PROGRAM UserMode
VAR

(*GapMode*)
	UserGapPositionNew:LREAL:=20;//target
	UserGapVelocityNew:LREAL:=1;//target
	UserGapPositionDisplay:LREAL;//current
	UserGapVelocityDisplay:LREAL;//current
(*ID taper mode*)
	UserTaperPositionNew:LREAL:=0;//target
	UserTaperVelocityNew:LREAL:=0.02;//target
	UserTaperPositionDisplay:LREAL;//current
	UserTaperPositionDisplayBLSide:LREAL;//current BeamLine
	UserTaperPositionActual:LREAL;//current
	UserTaperVelocityDisplay:LREAL;//target
	UserGapPositionDisplay_FromLeftTop:LREAL;
	UserGapPositionDisplay_FromLeftBottom:LREAL;
		//
	UserRightGapPositionNew:LREAL;
	UserRightGapVelocityNew:LREAL;
	UserRightGapPositionDisplay:LREAL;
	UserRightGapVelocityDisplay:LREAL;
	UserRightGapPositionDisplay_FromRightTop:LREAL;
	UserRightGapPositionDisplay_FromRightBottom:LREAL;
(*BL taper mode*)
	BLUserTaperPositionNew:LREAL:=0;//target
	BLUserTaperVelocityNew:LREAL:=0.02;//target
	BLUserTaperPositionDisplay:LREAL;//current
	//BLUserTaperPositionDisplayBLSide:LREAL;//current BeamLine
	BLUserTaperPositionActual:LREAL;//current
	BLUserTaperVelocityDisplay:LREAL;//target
	BLUserGapPositionDisplay_FromLeftTop:LREAL;
	BLUserGapPositionDisplay_FromLeftBottom:LREAL;
	//
	BLUserLeftGapPositionNew:LREAL;
	BLUserLeftGapVelocityNew:LREAL;
	BLUserLeftGapPositionDisplay:LREAL;
	BLUserLeftGapVelocityDisplay:LREAL;
	BLUserLeftGapPositionDisplay_FromLeftTop:LREAL;
	BLUserLeftGapPositionDisplay_FromLeftBottom:LREAL;
	BLUserRightGapPositionNew:LREAL;
	BLUserRightGapVelocityNew:LREAL;
	BLUserRightGapPositionDisplay:LREAL;
	BLUserRightGapVelocityDisplay:LREAL;
	BLUserRightGapPositionDisplay_FromRightTop:LREAL;
	BLUserRightGapPositionDisplay_FromRightBottom:LREAL;
(*PhaseUpper Move*)
	UserPhaseUpperPositionNew:LREAL:=0;//target
	UserPhaseUpperVelocityNew:LREAL:=0.5;//target
(*PhaseUpper Move*)
	UserPhaseLowerPositionNew:LREAL:=0;//target
	UserPhaseLowerVelocityNew:LREAL:=0.5;//target
	UserPhaseLowerPositionDisplay:LREAL;//current
	UserPhaseLowerVelocityDisplay:LREAL;//current
	//
	(*Gap move&Stop*)
	btn_UserGapMove:BOOL;
	btn_UserGapStop:BOOL;
	(*PhaseUpper Move&Stop*)
	btn_UserPhaseUpperMove:BOOL;
	btn_UserPhaseUpperStop:BOOL;
	(*PhaseLower Move&Stop*)
	btn_UserPhaseLowerMove:BOOL;
	btn_UserPhaseLowerStop:BOOL;
	(*Var*)
	fb_ton1:TON;
	fb_ton2:TON;
	fb_ton3:TON;
	fb_ton4:TON;
	fb_ton5:TON;
	fb_ton6:TON;
	(*Status*)
	State:DINT;
	Busy:BOOL;
	InitPowerDone:BOOL;
	InitCompensationDatasDone:BOOL;
	(*FB*)
	m_state: DINT;
	n_state: DINT;
	s_state: DINT;
	m_state_PhaseUpper: DINT;
	n_state_PhaseUpper: DINT;
	s_state_PhaseUpper: DINT;
	m_state_PhaseLower: DINT;
	n_state_PhaseLower: DINT;
	s_state_PhaseLower: DINT;
	(*¼ì²âµ½ÏÞÎ»£¬»Ö¸´Move×´Ì¬*)
	FTrig_ReachLS: F_TRIG;
	FTrig_ReachLS_PhaseUpper: F_TRIG;
	FTrig_ReachLS_PhaseLower: F_TRIG;
	FTrig_btn_GapMove: F_TRIG;
	GapOutRange: BOOL;
	(*PowerOff*)
	d_state: DINT;
	i: INT;
	j: INT;
	k: INT;
	moni_State:DINT;
	TargetPosLessThanCurrentPos:BOOL;
	TargetLTPosLessThanCurrentLTPos:BOOL;
	TargetRTPosLessThanCurrentRTPos:BOOL;
	TargetLBPosLessThanCurrentLBPos:BOOL;
	TargetRBPosLessThanCurrentRBPos:BOOL;
	PositiveMoving:BOOL;
	HysteresisMoving:BOOL;
	NoneHysteresisMoving:BOOL;
	(**)
	TargetPosLessThanCurrentPos_PhaseUpper:BOOL;
	PositiveMoving_PhaseUpper:BOOL;
	HysteresisMoving_PhaseUpper:BOOL;
	NoneHysteresisMoving_PhaseUpper:BOOL;
	TargetPosLessThanCurrentPos_PhaseLower:BOOL;
	PositiveMoving_PhaseLower:BOOL;
	HysteresisMoving_PhaseLower:BOOL;
	NoneHysteresisMoving_PhaseLower:BOOL;
	(*Spectroscopy scanning Mode*)
	IsSSMotionMode:BOOL;
	RegularMotionMode:BOOL;
	SSMotionMode:BOOL;
	SS_StepSize:LREAL:=0.001;
	SS_StepNumber:INT:=10;
	SS_StepVelocity:LREAL:=1;
	SS_Move:BOOL;
	SS_Stop:BOOL;
	SS_MoveState:DINT;
	SS_StopState:DINT;
	SS_currentStep:DINT:=0;
	SS_StepSystemTime_Begin:ARRAY[0..100] OF ULINT;
	SS_StepSystemTime_End:ARRAY[0..100] OF ULINT;
	SS_StepCountTime:ARRAY[0..100] OF ULINT;
	SS_TimeCountBegin:BOOL;
	m: INT;
	SS_TON: TON;
	StepEachTime:TIME;
	StepEachTime_ms:INT:=1000;//ms
	SS_OTSTRUCT :OTSTRUCT ;
	SS_StartPositionDisplay:LREAL;
	RTRG_SS_StartPositionDisplay:R_TRIG;
	SS_InitStartPositionDone:BOOL;
	
	//
	min_SS_StepSize	: LREAL:=0;
	max_SS_StepSize	: LREAL:=200;
	inRange_SS_StepSize	: BOOL;
	//
	min_SS_StepNumber	: INT:=1;
	max_SS_StepNumber	: INT:=1000;
	inRange_SS_StepNumber	: BOOL;
	//
	min_SS_StepVelocity:LREAL:=0;
	max_SS_StepVelocity:LREAL:=1;
	inRange_SS_StepVelocity:BOOL;
	//
	min_StepEachTime_ms:INT:=100;
	max_StepEachTime_ms:INT:=10000;
	inRange_StepEachTime_ms:BOOL;
	l: INT;
	Threshold_UserTopPos_PLC: LREAL;
	Threshold_UserTopVelo_PLC: LREAL;
	Threshold_UserBottomPos_PLC: LREAL;
	Threshold_UserBottomVelo_PLC: LREAL;
	Threshold_UserLeftPos_PLC: LREAL;
	Threshold_UserLeftVelo_PLC: LREAL;
	Threshold_UserRightPos_PLC: LREAL;
	Threshold_UserRightVelo_PLC: LREAL;
	testa: BOOL;
	testb: BOOL;
	Threshold_GapChangeFlag: LREAL;
	Threshold_TaperChangeFlag: LREAL;
	TaperAndGapSafetyfactor: LREAL:=1;
	//GapPhase Chain protection
	GapPhase_ChainProtection_On:BOOL;
	GapPhase_ChainProtection_MaxGapValue: LREAL;
	//
	//Global Chain protection-MPS
	Global_ChainProtection_MPS_StorageRingReady:BOOL;
	Global_ChainProtection_MPS_On: BOOL;
	Global_ChainProtection_MPS_MaxGapValue: LREAL;
	Global_ChainProtection_MPS_MoveVelocity: LREAL;
	Global_ChainProtection_MPS_Done: BOOL;
	//Global_ChainProtection_Error: BOOL;
	//Global_ChainProtection_ErrorID: INT;
	//Global_ChainProtection_ErrorDescription: STRING;
	Global_ChainProtection_MPS_ManualOperation:BOOL:=TRUE;
	Global_ChainProtection_MPS_FTRIG:F_TRIG;
	Global_ChainProtection_MPS_FTRIG_Manul:F_TRIG;
	Global_ChainProtection_MPS_TON:TON;
	Global_ChainProtection_MPS_Triggered:BOOL;
	Global_ChainProtection_MPS_In:BOOL;
	Global_ChainProtection_MPS_In1 AT%I* :BOOL;//下降沿表示触发,EL1008
	Global_ChainProtection_MPS_In2 AT%I* :BOOL;
	Global_ChainProtection_MPS_State:DINT;
	Global_ChainProtection_MPS_Out1 AT%Q* :BOOL;//上升沿标识到达最大间隙，连锁保护成功,EL2624
	Global_ChainProtection_MPS_Out2 AT%Q* :BOOL;
	Global_ChainProtection_MPS_TON_Stop2Move:TON;
	Global_ChainProtection_MPS_TON_Stop2Move_InTaperMode:TON;
	Global_ChainProtection_MPS_TON_Power2Move:TON;
	//Global Chain protection-EPS
	Global_ChainProtection_EPS_BeamLineReady:BOOL;
	Global_ChainProtection_EPS_On: BOOL;
	Global_ChainProtection_EPS_MaxGapValue: LREAL;
	Global_ChainProtection_EPS_MoveVelocity: LREAL;
	Global_ChainProtection_EPS_Done: BOOL;
	//Global_ChainProtection_Error: BOOL;
	//Global_ChainProtection_ErrorID: INT;
	//Global_ChainProtection_ErrorDescription: STRING;
	Global_ChainProtection_EPS_ManualOperation:BOOL:=TRUE;
	Global_ChainProtection_EPS_FTRIG:F_TRIG;
	Global_ChainProtection_EPS_FTRIG_Manul:F_TRIG;
	Global_ChainProtection_EPS_TON:TON;
	Global_ChainProtection_EPS_Triggered:BOOL;
	Global_ChainProtection_EPS_In:BOOL;
	Global_ChainProtection_EPS_In1 AT%I* :BOOL;//下降沿表示触发,EL1124
	Global_ChainProtection_EPS_In2 AT%I* :BOOL;
	Global_ChainProtection_EPS_State:DINT;
	Global_ChainProtection_EPS_Out1 AT%Q* :BOOL;//上升沿标识到达最大间隙，连锁保护成功,EL2124
	Global_ChainProtection_EPS_Out2 AT%Q* :BOOL;
	Global_ChainProtection_EPS_TON_Stop2Move:TON;
	Global_ChainProtection_EPS_TON_Stop2Move_InTaperMode:TON;
	Global_ChainProtection_EPS_TON_Power2Move:TON;
	
	Threshold_motorsTargetPosCalculate: LREAL;
	LeftTopLinPositionNewTemp: LREAL;
	RightTopLinPositionNewTemp: LREAL;
	LeftBottomLinPositionNewTemp: LREAL;
	RightBottomLinPositionNewTemp: LREAL;
	UserPhaseUpperPositionNewTemp: LREAL;
	UserPhaseLowerPositionNewTemp: LREAL;
	
	//OneKeyToMaxGap
	btn_OneKeyToMaxGap:BOOL;
	OneKeyToMaxGap_RTRIG:R_TRIG;
	OneKeyToMaxGap_TON:TON;
	OneKeyToMaxGap_Triggered:BOOL;
	OneKeyToMaxGap_State:DINT;
	OneKeyToMaxGap_TON_Stop2Move:TON;
	OneKeyToMaxGap_TON_Stop2Move_InTaperMode:TON;
	OneKeyToMaxGap_TON_Power2Move:TON;
	OneKeyToMaxGap_Done:BOOL;
	
		//BLTaper
	CurrentTaperInit: LREAL;
	L_HalfGirder:LREAL:=2500;
	L_Center2Motor:LREAL:=1375;
	//
	trig_TaperOrNot: R_TRIG;
	trig_BLTaperOrNot: R_TRIG;
	
	//
	//零位特殊走法
	//
	(*Upper*)
    // 零位特殊走法总开关。TRUE 启用；FALSE 关闭，关闭后直接按原 m/n 正常逻辑运行。
    EnableZeroPre_PhaseUpper : BOOL := TRUE;

    // 判断“当前位置在零附近”的范围。例如当前位置绝对值 <= 0.01mm 认为在零附近。
    ZeroNearThreshold_PhaseUpper : LREAL := 0.3;

    // 原来的 +/-1mm 边界，做成变量，后续可以改成 +/-0.5mm、+/-2mm 等。
    ZeroBoundary_PhaseUpper : LREAL := 1.5;

    // 零位附近特殊慢速，原来的 0.1mm/s，做成变量。
    ZeroSlowVelocity_PhaseUpper : LREAL := 0.1;

    // TRUE 表示当前正在执行零位预走状态机，此时屏蔽原 m/n 正常逻辑。
    ZeroPreMoving_PhaseUpper : BOOL := FALSE;

    // TRUE 表示本次 Move 的零位预走已经完成，下一步允许进入原 m/n 正常逻辑；正常完成或 Stop 时必须清 FALSE。
    ZeroPreDone_PhaseUpper : BOOL := FALSE;

    // TRUE 表示目标就在 +/-ZeroBoundary_PhaseUpper 内，此时只需要慢速直接走到目标，不再进入原 m/n 正常逻辑。
    ZeroDirectMove_PhaseUpper : BOOL := FALSE;

    // 零位预走专用状态。
    z_state_PhaseUpper : INT := 0;

    // 零位预走第一段目标：目标超过边界时为 +ZeroBoundary/-ZeroBoundary；目标在边界内时为最终目标。
    ZeroPreTarget_PhaseUpper : LREAL := 0.0;

    // 锁存本次 Move 的最终目标，避免零位慢速段期间用户改输入导致最终目标漂移。
    ZeroFinalTarget_PhaseUpper : LREAL := 0.0;

    // 锁存本次 Move 的用户速度，零位预走之后原 m/n 逻辑使用这个速度。
    ZeroFinalVelocity_PhaseUpper : LREAL := 0.0;

    // 原 m/n 正常逻辑当前使用的目标；零位预走后用 ZeroFinalTarget_PhaseUpper，否则用 UserPhaseUpperPositionNew。
    ActiveTarget_PhaseUpper : LREAL := 0.0;

    // 原 m/n 正常逻辑当前使用的速度；零位预走后用 ZeroFinalVelocity_PhaseUpper，否则用 UserPhaseUpperVelocityNew。
    ActiveVelocity_PhaseUpper : LREAL := 0.0;
	
	(*Lower*)
	
    // 零位特殊走法总开关。TRUE 启用；FALSE 关闭，关闭后直接按原 m/n 正常逻辑运行。
    EnableZeroPre_PhaseLower : BOOL := TRUE;

    // 判断“当前位置在零附近”的范围。例如当前位置绝对值 <= 0.01mm 认为在零附近。
    ZeroNearThreshold_PhaseLower : LREAL := 0.3;

    // 原来的 +/-1mm 边界，做成变量，后续可以改成 +/-0.5mm、+/-2mm 等。
    ZeroBoundary_PhaseLower : LREAL := 1.5;

    // 零位附近特殊慢速，原来的 0.1mm/s，做成变量。
    ZeroSlowVelocity_PhaseLower : LREAL := 0.1;

    // TRUE 表示当前正在执行零位预走状态机，此时屏蔽原 m/n 正常逻辑。
    ZeroPreMoving_PhaseLower : BOOL := FALSE;

    // TRUE 表示本次 Move 的零位预走已经完成，下一步允许进入原 m/n 正常逻辑；正常完成或 Stop 时必须清 FALSE。
    ZeroPreDone_PhaseLower : BOOL := FALSE;

    // TRUE 表示目标就在 +/-ZeroBoundary_PhaseLower 内，此时只需要慢速直接走到目标，不再进入原 m/n 正常逻辑。
    ZeroDirectMove_PhaseLower : BOOL := FALSE;

    // 零位预走专用状态。
    z_state_PhaseLower : INT := 0;

    // 零位预走第一段目标：目标超过边界时为 +ZeroBoundary/-ZeroBoundary；目标在边界内时为最终目标。
    ZeroPreTarget_PhaseLower : LREAL := 0.0;

    // 锁存本次 Move 的最终目标，避免零位慢速段期间用户改输入导致最终目标漂移。
    ZeroFinalTarget_PhaseLower : LREAL := 0.0;

    // 锁存本次 Move 的用户速度，零位预走之后原 m/n 逻辑使用这个速度。
    ZeroFinalVelocity_PhaseLower : LREAL := 0.0;

    // 原 m/n 正常逻辑当前使用的目标；零位预走后用 ZeroFinalTarget_PhaseLower，否则用 UserPhaseLowerPositionNew。
    ActiveTarget_PhaseLower : LREAL := 0.0;

    // 原 m/n 正常逻辑当前使用的速度；零位预走后用 ZeroFinalVelocity_PhaseLower，否则用 UserPhaseLowerVelocityNew。
    ActiveVelocity_PhaseLower : LREAL := 0.0;
 
	
END_VAR

IF NOT PositionBiasDone THEN
	RETURN;
END_IF
IF NOT loadParametersDone THEN
	RETURN;
END_IF
(*btn_Power On/Off*)
IF btn_Power AND st_Power=0 THEN
	btn_PowerOn:=TRUE;
	btn_Power:=FALSE;
END_IF
IF btn_Power AND st_Power=1 THEN
	btn_PowerOff:=TRUE;
	btn_Power:=FALSE;
END_IF
IF btn_PowerOn THEN
	A_PowerOn();
END_IF
IF btn_PowerOff THEN
	A_PowerOff();
END_IF

(*检查couple状态，不允许couple*)
A_CheckCoupleStatus();

(*监控四轴位置速度等*)
A_MonitoringAllAxis();

(*补偿数据处理*)
A_InitCompensationData();

(*目标位置和速度保护*)
A_CheckMotorsPos();


(*常规磁间隙开合*)
//IF RegularMotionMode AND NOT SSMotionMode THEN
A_RegularMotion();
//END_IF
(*PhaseUpper运动*)
A_PhaseUpperMotion();
(*PhaseLower运动*)
A_PhaseLowerMotion();
(*Spectroscopy scanning Mode*)
IF IsSSMotionMode THEN
	SSMotionMode:=TRUE;
	RegularMotionMode:=FALSE;
ELSE
	SSMotionMode:=FALSE;
	RegularMotionMode:=TRUE;
END_IF
IF	SSMotionMode AND NOT RegularMotionMode THEN
	A_SpectroscopyScanningMotion();
END_IF
(*GlobalChainProtection*)
A_GlobalChainProtection_EPS();
A_GlobalChainProtection_MPS();
(*A_OneKeyToMaxGap*)
A_OneKeyToMaxGap();

ACTION A_CheckCoupleStatus:
IF NOT btn_PowerOff THEN
	IF st_Power=1 AND st_Couple<>0THEN
		Error:=TRUE;
		ErrorID:=501;
		LeftTopLinMoveIndicator:=0;
		RightTopLinMoveIndicator:=0;
		LeftBottomLinMoveIndicator:=0;
		RightBottomLinMoveIndicator:=0;
		FB_PlcEmergencyStop();
		LED_Error:=TRUE;
		ErrorDescription:='couple stutas error';
	END_IF
END_IF
END_ACTION

ACTION A_CheckMotorsPos:
//
//目标位置速度超出阈值判断
//
//gap posiion
IF UserGapPositionNew<min_UserGapPositionNew OR UserGapPositionNew>max_UserGapPositionNew THEN
	inRange_UserGapPositionNew:=FALSE;
END_IF
IF UserGapPositionNew>=min_UserGapPositionNew AND UserGapPositionNew<=max_UserGapPositionNew THEN
	inRange_UserGapPositionNew:=TRUE;
END_IF
//gap velocity
IF UserGapVelocityNew<min_UserGapVelocityNew OR UserGapVelocityNew>max_UserGapVelocityNew THEN
	inRange_UserGapVelocityNew:=FALSE;
END_IF
IF UserGapVelocityNew>=min_UserGapVelocityNew AND UserGapVelocityNew<=max_UserGapVelocityNew THEN
	inRange_UserGapVelocityNew:=TRUE;
END_IF
//taper position
IF UserTaperPositionNew<min_UserTaperPositionNew OR UserTaperPositionNew>max_UserTaperPositionNew THEN
	inRange_UserTaperPositionNew:=FALSE;
END_IF
IF UserTaperPositionNew>=min_UserTaperPositionNew AND UserTaperPositionNew<=max_UserTaperPositionNew THEN
	inRange_UserTaperPositionNew:=TRUE;
END_IF
//taper velocity
IF UserTaperVelocityNew<min_UserTaperVelocityNew OR UserTaperVelocityNew>max_UserTaperVelocityNew THEN
	inRange_UserTaperVelocityNew:=FALSE;
END_IF
IF UserTaperVelocityNew>=min_UserTaperVelocityNew AND UserTaperVelocityNew<=max_UserTaperVelocityNew THEN
	inRange_UserTaperVelocityNew:=TRUE;
END_IF
//
//PhaseUpper posiion
IF UserPhaseUpperPositionNew<min_UserPhaseUpperPositionNew OR UserPhaseUpperPositionNew>max_UserPhaseUpperPositionNew THEN
	inRange_UserPhaseUpperPositionNew:=FALSE;
END_IF
IF UserPhaseUpperPositionNew>=min_UserPhaseUpperPositionNew AND UserPhaseUpperPositionNew<=max_UserPhaseUpperPositionNew THEN
	inRange_UserPhaseUpperPositionNew:=TRUE;
END_IF
//gap velocity
IF UserPhaseUpperVelocityNew<min_UserPhaseUpperVelocityNew OR UserPhaseUpperVelocityNew>max_UserPhaseUpperVelocityNew THEN
	inRange_UserPhaseUpperVelocityNew:=FALSE;
END_IF
IF UserPhaseUpperVelocityNew>=min_UserPhaseUpperVelocityNew AND UserPhaseUpperVelocityNew<=max_UserPhaseUpperVelocityNew THEN
	inRange_UserPhaseUpperVelocityNew:=TRUE;
END_IF
//PhaseLower posiion
IF UserPhaseLowerPositionNew<min_UserPhaseLowerPositionNew OR UserPhaseLowerPositionNew>max_UserPhaseLowerPositionNew THEN
	inRange_UserPhaseLowerPositionNew:=FALSE;
END_IF
IF UserPhaseLowerPositionNew>=min_UserPhaseLowerPositionNew AND UserPhaseLowerPositionNew<=max_UserPhaseLowerPositionNew THEN
	inRange_UserPhaseLowerPositionNew:=TRUE;
END_IF
//gap velocity
IF UserPhaseLowerVelocityNew<min_UserPhaseLowerVelocityNew OR UserPhaseLowerVelocityNew>max_UserPhaseLowerVelocityNew THEN
	inRange_UserPhaseLowerVelocityNew:=FALSE;
END_IF
IF UserPhaseLowerVelocityNew>=min_UserPhaseLowerVelocityNew AND UserPhaseLowerVelocityNew<=max_UserPhaseLowerVelocityNew THEN
	inRange_UserPhaseLowerVelocityNew:=TRUE;
END_IF
//SS Mode
IF SS_StepSize<min_SS_StepSize OR SS_StepSize>max_SS_StepSize THEN
	inRange_SS_StepSize:=FALSE;
END_IF
IF SS_StepSize>=min_SS_StepSize AND SS_StepSize<=max_SS_StepSize THEN
	inRange_SS_StepSize:=TRUE;
END_IF
IF SS_StepNumber<min_SS_StepNumber OR SS_StepNumber>max_SS_StepNumber THEN
	inRange_SS_StepNumber:=FALSE;
END_IF
IF SS_StepNumber>=min_SS_StepNumber AND SS_StepNumber<=max_SS_StepNumber THEN
	inRange_SS_StepNumber:=TRUE;
END_IF
IF SS_StepVelocity<min_SS_StepVelocity OR SS_StepVelocity>max_SS_StepVelocity THEN
	inRange_SS_StepVelocity:=FALSE;
END_IF
IF SS_StepVelocity>=min_SS_StepVelocity AND SS_StepVelocity<=max_SS_StepVelocity THEN
	inRange_SS_StepVelocity:=TRUE;
END_IF
IF StepEachTime_ms<min_StepEachTime_ms OR StepEachTime_ms>max_StepEachTime_ms THEN
	inRange_StepEachTime_ms:=FALSE;
END_IF
IF StepEachTime_ms>=min_StepEachTime_ms AND StepEachTime_ms<=max_StepEachTime_ms THEN
	inRange_StepEachTime_ms:=TRUE;
END_IF


//
//输入速度和位置保护
//
IF btn_UserGapMove  AND NOT SSMotionMode AND RegularMotionMode THEN
	IF NOT inRange_UserGapPositionNew THEN
		btn_UserGapStop:=TRUE;
		btn_UserGapMove:=FALSE;
		Error:=TRUE;
		ErrorId:=801;
		ErrorDescription:='target Gap position out of range,please check';
		RETURN;
	ELSE
		//btn_UserGapStop:=FALSE;
		Error:=FALSE;
		ErrorId:=0;
		ErrorDescription:='';	
	END_IF
	IF NOT inRange_UserGapVelocityNew THEN
		btn_UserGapStop:=TRUE;
		btn_UserGapMove:=FALSE;
		Error:=TRUE;
		ErrorId:=802;
		ErrorDescription:='target Gap velocity out of range,please check';
		RETURN;
	ELSE
		//btn_UserGapStop:=FALSE;
		Error:=FALSE;
		ErrorId:=0;
		ErrorDescription:='';
	END_IF
END_IF

//
//运动过程中，监控目标位置速度
//
IF moveStatusAnyAxis THEN
	IF NOT inRange_UserGapPositionNew THEN
		btn_UserGapStop:=TRUE;
		Error:=TRUE;
		ErrorId:=805;
		ErrorDescription:='target Gap position out of range in moving process!';
		FB_PlcEmergencyStop();
	END_IF
	IF NOT inRange_UserGapVelocityNew THEN
		btn_UserGapStop:=TRUE;
		Error:=TRUE;
		ErrorId:=806;
		ErrorDescription:='target Gap velocity out of range in moving process!';
		FB_PlcEmergencyStop();
	END_IF
END_IF
//
//运动过程中，监控每一个轴的目标位置，目标位置若超出阈值，Emergency
//
IF moveStatusAnyAxis THEN
	IF NOT TaperOrNot THEN
		IF LeftTopLinPositionNew<min_UserLEProtectionGapPosition/2 OR LeftTopLinPositionNew>max_UserLEProtectionGapPosition/2 THEN
			btn_UserGapStop:=TRUE;
			Error:=TRUE;
			ErrorId:=809;
			ErrorDescription:='target LeftTop position out of range in moving process!';
			FB_PlcEmergencyStop();
		END_IF
		IF RightTopLinPositionNew<min_UserLEProtectionGapPosition/2 OR RightTopLinPositionNew>max_UserLEProtectionGapPosition/2 THEN
			btn_UserGapStop:=TRUE;
			Error:=TRUE;
			ErrorId:=810;
			ErrorDescription:='target RightTop velocity out of range in moving process!';
			FB_PlcEmergencyStop();
		END_IF
		IF LeftBottomLinPositionNew<min_UserLEProtectionGapPosition/2 OR LeftBottomLinPositionNew>max_UserLEProtectionGapPosition/2 THEN
			btn_UserGapStop:=TRUE;
			Error:=TRUE;
			ErrorId:=812;
			ErrorDescription:='target LeftBottom Position out of range in moving process!';
			FB_PlcEmergencyStop();
		END_IF
		IF RightBottomLinPositionNew<min_UserLEProtectionGapPosition/2 OR RightBottomLinPositionNew>max_UserLEProtectionGapPosition/2 THEN
			btn_UserGapStop:=TRUE;
			Error:=TRUE;
			ErrorId:=813;
			ErrorDescription:='target RightBottom Position out of range in moving process!';
			FB_PlcEmergencyStop();
		END_IF
	ELSE//Taper状态的保护
		;//Taper状态下，不用监控四轴位置，只需要监控目标Taper位置。在上面已经保护
	END_IF
END_IF
END_ACTION

ACTION A_GlobalChainProtection_EPS:
//硬线输入定义
Global_ChainProtection_EPS_In:=Global_ChainProtection_EPS_In1 AND Global_ChainProtection_EPS_In2;
//硬线输出定义
Global_ChainProtection_EPS_Out1:=Global_ChainProtection_EPS_Done;
Global_ChainProtection_EPS_Out2:=Global_ChainProtection_EPS_Done;
//总开关
IF NOT Global_ChainProtection_EPS_On THEN
	RETURN;
END_IF
//判断插入件状态，是否就位
//IF NOT IDControlReady THEN
//	Global_ChainProtection_EPS_Done:=FALSE;
//	Error:= TRUE;
//	ErrorID:= 1501;
//	ErrorDescription:='ID NOT READY!';
//	RETURN;
//END_IF
//判断储存环是否给出就位信号，暂时由参数表给出TRUE，最终将由IOC接受PV
IF 	NOT Global_ChainProtection_EPS_BeamLineReady THEN
	Global_ChainProtection_EPS_Done:=FALSE;
	Error:= TRUE;
	ErrorID:= 1503;
	ErrorDescription:='Global_ChainProtection_EPS_BeamLineReady NOT Ready';
	RETURN;
END_IF
//
//全局连锁保护程序开始
//
//0.检测到下降沿，触发
//1.判断电机是否在开启状态,没有就打开电源
//2.判断是否在Moving状态,若有就Stop
//3.将磁间隙打开到至最大阈值
//4.到位后给出反馈，且安全PLC触发
Global_ChainProtection_EPS_FTRIG(CLK:=Global_ChainProtection_EPS_In);
IF Global_ChainProtection_EPS_FTRIG.Q THEN
	Global_ChainProtection_EPS_Triggered:=TRUE;
END_IF
Global_ChainProtection_EPS_FTRIG_Manul(CLK:=Global_ChainProtection_EPS_ManualOperation);
IF Global_ChainProtection_EPS_FTRIG_Manul.Q THEN
	Global_ChainProtection_EPS_Triggered:=TRUE;
END_IF
IF Global_ChainProtection_EPS_Triggered THEN
	CASE Global_ChainProtection_EPS_State OF
		0://1.判断电机是否在开启状态,没有就打开电源
			IF st_Power=1 THEN
				Global_ChainProtection_EPS_State:=1;
			ELSE
				btn_PowerOn:=TRUE;
				IF btn_PowerOn THEN
					A_PowerOn();
				END_IF
			END_IF
		1://1.判断是否在谱学扫描模式，如果是，则切换回正常运动模式
			IF IsSSMotionMode THEN
				SS_Stop:=TRUE;
				IsSSMotionMode:=FALSE;
			END_IF
			Global_ChainProtection_EPS_State:=2;
		2://判断是否在taper，如果在taper,则判断是否在运动，如果是，则停止运动,0.5sh后，转入下一步
			IF TaperOrNot THEN
				IF moveStatusLeftTop OR moveStatusRightTop OR moveStatusLeftBottom OR moveStatusRightBottom THEN
					btn_UserGapStop:=TRUE;
				ELSE
					Global_ChainProtection_EPS_TON_Stop2Move_InTaperMode(PT:=T#0.5S);
					Global_ChainProtection_EPS_TON_Stop2Move_InTaperMode.IN:=TRUE;
					IF Global_ChainProtection_EPS_TON_Stop2Move_InTaperMode.Q THEN
						TaperOrNot:=FALSE;//关闭taper模式
						Global_ChainProtection_EPS_State:=3;
					END_IF
				END_IF
			ELSE
				Global_ChainProtection_EPS_State:=3;
			END_IF
		3://3.判断是否在Moving状态,若有就Stop.Taper模式已处理完，此处开始走正常GAP开合逻辑
			IF moveStatusLeftTop OR moveStatusRightTop OR moveStatusLeftBottom OR moveStatusRightBottom THEN
				btn_UserGapStop:=TRUE;
			ELSE
				Global_ChainProtection_EPS_TON_Stop2Move(PT:=T#0.5S);
				Global_ChainProtection_EPS_TON_Stop2Move.IN:=TRUE;
				IF Global_ChainProtection_EPS_TON_Stop2Move.Q THEN
					Global_ChainProtection_EPS_State:=4;
				END_IF
			END_IF
		4://当前磁间隙如何和最大磁间隙差别不大，不超过0.1，则直接保护
			IF ABS(UserGapPositionDisplay-Global_ChainProtection_EPS_MaxGapValue)<=0.1 THEN
				Global_ChainProtection_EPS_Done:=TRUE;
				Plc_EmergencyStop:=FALSE;	
				Error:=TRUE;
				ErrorID:=1506;
				ErrorDescription:='EPS Triggered,but ABS(UserGapPositionDisplay-Global_ChainProtection_EPS_MaxGapValue)<=0.1 ';	
			ELSE
				Global_ChainProtection_EPS_State:=5;
			END_IF
		5://5.将磁间隙打开到至最大阈值
			Global_ChainProtection_EPS_TON(PT:=INT_TO_TIME(LREAL_TO_INT(Global_ChainProtection_EPS_MaxGapValue/Global_ChainProtection_EPS_MoveVelocity+30))*1000);
			Global_ChainProtection_EPS_TON.IN:=TRUE;
			Global_ChainProtection_EPS_TON_Power2Move(PT:=T#0.1S);
			Global_ChainProtection_EPS_TON_Power2Move.IN:=TRUE;
			UserGapPositionNew:=Global_ChainProtection_EPS_MaxGapValue;
			UserGapVelocityNew:=Global_ChainProtection_EPS_MoveVelocity;
			btn_UserGapMove:=TRUE;
			IF Global_ChainProtection_EPS_TON_Power2Move.Q THEN
				IF FB_MOVE.BCGapDone THEN
					Global_ChainProtection_EPS_State:=88;
				END_IF
			END_IF
			IF Global_ChainProtection_EPS_TON.Q THEN//如果150s后，还没有运动到指定gap，则报错
				Global_ChainProtection_EPS_State:=-100;
			END_IF
		88://6.到位后给出反馈，且安全PLC触发
			Global_ChainProtection_EPS_Done:=TRUE;
			Plc_EmergencyStop:=FALSE;	
			Error:=TRUE;
			ErrorID:=1504;
			ErrorDescription:='Global_ChainProtection_EPS Triggered ';	
		-100:
			Global_ChainProtection_EPS_Done:=FALSE;
			Error:=TRUE;
			ErrorID:=1505;
			ErrorDescription:='NOT MOVING TO MAXGAP';
	END_CASE
END_IF
END_ACTION

ACTION A_GlobalChainProtection_MPS:
//硬线输入定义
Global_ChainProtection_MPS_In:=Global_ChainProtection_MPS_In1 AND Global_ChainProtection_MPS_In2;
//硬线输出定义
Global_ChainProtection_MPS_Out1:=Global_ChainProtection_MPS_Done;
Global_ChainProtection_MPS_Out2:=Global_ChainProtection_MPS_Done;
//总开关
IF NOT Global_ChainProtection_MPS_On THEN
	RETURN;
END_IF
//判断插入件状态，是否就位
//IF NOT IDControlReady THEN
//	Global_ChainProtection_MPS_Done:=FALSE;
//	Error:= TRUE;
//	ErrorID:= 1401;
//	ErrorDescription:='ID NOT READY!';
//	RETURN;
//END_IF
//判断储存环是否给出就位信号，暂时由参数表给出TRUE，最终将由IOC接受PV
IF 	NOT Global_ChainProtection_MPS_StorageRingReady THEN
	Global_ChainProtection_MPS_Done:=FALSE;
	Error:= TRUE;
	ErrorID:= 1403;
	ErrorDescription:='StorageRingChainProtection NOT Ready';
	RETURN;
END_IF
//
//全局连锁保护程序开始
//
//0.检测到下降沿，触发
//1.判断电机是否在开启状态,没有就打开电源
//2.判断是否在Moving状态,若有就Stop
//3.将磁间隙打开到至最大阈值
//4.到位后给出反馈，且安全PLC触发
Global_ChainProtection_MPS_FTRIG(CLK:=Global_ChainProtection_MPS_In);
IF Global_ChainProtection_MPS_FTRIG.Q THEN
	Global_ChainProtection_MPS_Triggered:=TRUE;
END_IF
Global_ChainProtection_MPS_FTRIG_Manul(CLK:=Global_ChainProtection_MPS_ManualOperation);
IF Global_ChainProtection_MPS_FTRIG_Manul.Q THEN
	Global_ChainProtection_MPS_Triggered:=TRUE;
END_IF
IF Global_ChainProtection_MPS_Triggered THEN
	CASE Global_ChainProtection_MPS_State OF
		0://1.判断电机是否在开启状态,没有就打开电源
			IF st_Power=1 THEN
				Global_ChainProtection_MPS_State:=1;
			ELSE
				btn_PowerOn:=TRUE;
				IF btn_PowerOn THEN
					A_PowerOn();
				END_IF
			END_IF
		1://1.判断是否在谱学扫描模式，如果是，则切换回正常运动模式
			IF IsSSMotionMode THEN
				SS_Stop:=TRUE;
				IsSSMotionMode:=FALSE;
			END_IF
			Global_ChainProtection_MPS_State:=2;
		2://判断是否在taper，如果在taper,则判断是否在运动，如果是，则停止运动,0.5sh后，转入下一步
			IF TaperOrNot THEN
				IF moveStatusLeftTop OR moveStatusRightTop OR moveStatusLeftBottom OR moveStatusRightBottom THEN
					btn_UserGapStop:=TRUE;
				ELSE
					Global_ChainProtection_MPS_TON_Stop2Move_InTaperMode(PT:=T#0.5S);
					Global_ChainProtection_MPS_TON_Stop2Move_InTaperMode.IN:=TRUE;
					IF Global_ChainProtection_MPS_TON_Stop2Move_InTaperMode.Q THEN
						TaperOrNot:=FALSE;//关闭taper模式
						Global_ChainProtection_MPS_State:=3;
					END_IF
				END_IF
			ELSE
				Global_ChainProtection_MPS_State:=3;
			END_IF
		3://3.判断是否在Moving状态,若有就Stop.Taper模式已处理完，此处开始走正常GAP开合逻辑
			IF moveStatusLeftTop OR moveStatusRightTop OR moveStatusLeftBottom OR moveStatusRightBottom THEN
				btn_UserGapStop:=TRUE;
			ELSE
				Global_ChainProtection_MPS_TON_Stop2Move(PT:=T#0.5S);
				Global_ChainProtection_MPS_TON_Stop2Move.IN:=TRUE;
				IF Global_ChainProtection_MPS_TON_Stop2Move.Q THEN
					Global_ChainProtection_MPS_State:=4;
				END_IF
			END_IF
		4://当前磁间隙如何和最大磁间隙差别不大，不超过0.1，则直接保护
			IF ABS(UserGapPositionDisplay-Global_ChainProtection_MPS_MaxGapValue)<=0.1 THEN
				Global_ChainProtection_MPS_Done:=TRUE;
				Plc_EmergencyStop:=FALSE;	
				Error:=TRUE;
				ErrorID:=1406;
				ErrorDescription:='MPS Triggered,but ABS(UserGapPositionDisplay-Global_ChainProtection_MPS_MaxGapValue)<=0.1 ';	
			ELSE
				Global_ChainProtection_MPS_State:=5;
			END_IF
		5://5.将磁间隙打开到至最大阈值
			Global_ChainProtection_MPS_TON(PT:=INT_TO_TIME(LREAL_TO_INT(Global_ChainProtection_MPS_MaxGapValue/Global_ChainProtection_MPS_MoveVelocity+30))*1000);
			Global_ChainProtection_MPS_TON.IN:=TRUE;
			Global_ChainProtection_MPS_TON_Power2Move(PT:=T#0.1S);
			Global_ChainProtection_MPS_TON_Power2Move.IN:=TRUE;
			UserGapPositionNew:=Global_ChainProtection_MPS_MaxGapValue;
			UserGapVelocityNew:=Global_ChainProtection_MPS_MoveVelocity;
			btn_UserGapMove:=TRUE;
			IF Global_ChainProtection_MPS_TON_Power2Move.Q THEN
				IF FB_MOVE.BCGapDone THEN
					Global_ChainProtection_MPS_State:=88;
				END_IF
			END_IF
			IF Global_ChainProtection_MPS_TON.Q THEN//如果150s后，还没有运动到指定gap，则报错
				Global_ChainProtection_MPS_State:=-100;
			END_IF
		88://6.到位后给出反馈，且安全PLC触发
			Global_ChainProtection_MPS_Done:=TRUE;
			Plc_EmergencyStop:=FALSE;	
			Error:=TRUE;
			ErrorID:=1404;
			ErrorDescription:='Global_ChainProtection_MPS Triggered ';	
		-100:
			Global_ChainProtection_MPS_Done:=FALSE;
			Error:=TRUE;
			ErrorID:=1405;
			ErrorDescription:='NOT MOVING TO MAXGAP';
	END_CASE
END_IF
END_ACTION

ACTION A_InitCompensationData:
(*补偿开始*)
IF USE_SingleAxis_Compensation THEN
	//
	//1.目标位置解算
	//
	(*通过补偿表解算四轴目标位置*)
	//左轴位置由Gap定，右轴位置由右gap定。右gap值=左gap+taper。taper模式和非taper模式一样，非taper模式只是一种特例存在
	//左轴目标位置解算
	IF NOT TaperOrNot THEN
		UserTaperPositionNew:=0;
		//UserTaperPositionDisplay:=0;
	END_IF
	UserRightGapPositionNew:=UserGapPositionNew+UserTaperPositionNew;
	//左轴目标位置解算
	FOR	i:= 1 TO 17 DO
			IF UserGapPositionNew/2<M_Compensation[i+1].Encoder AND UserGapPositionNew/2>=M_Compensation[i].Encoder THEN
				IF i<>18 THEN
					LeftTopLinPositionNew:=(((UserGapPositionNew/2-M_Compensation[i].Encoder)*(M_Compensation[i+1].LeftTop-M_Compensation[i].LeftTop))
							/(M_Compensation[i+1].Encoder-M_Compensation[i].Encoder))+M_Compensation[i].LeftTop;
					LeftBottomLinPositionNew:=(((UserGapPositionNew/2-M_Compensation[i].Encoder)*(M_Compensation[i+1].LeftBottom-M_Compensation[i].LeftBottom))
							/(M_Compensation[i+1].Encoder-M_Compensation[i].Encoder))+M_Compensation[i].LeftBottom;
					M_CompensationNumber:=i;
					InitCompensationDatasDone:=TRUE;
				ELSIF i=18 AND UserGapPositionNew/2=M_Compensation[i].Encoder THEN		(*Gap=14µÄÌØÊâÇé¿ö*)
					(**)
					LeftTopLinPositionNew:=M_Compensation[i].LeftTop;
					LeftBottomLinPositionNew:=M_Compensation[i].LeftBottom;
					M_CompensationNumber:=i;
					InitCompensationDatasDone:=TRUE;
				ELSE
					LeftTopLinPositionNew:=UserGapPositionNew/2;
					LeftBottomLinPositionNew:=UserGapPositionNew/2;
					M_CompensationNumber:=i;
					InitCompensationDatasDone:=TRUE;
				END_IF
			END_IF
	END_FOR
	//右轴目标位置解算
	FOR	j:= 1 TO 17 DO
		IF UserRightGapPositionNew/2<M_Compensation[j+1].Encoder AND UserRightGapPositionNew/2>=M_Compensation[j].Encoder THEN
			IF j<>18 THEN
				RightTopLinPositionNew:=(((UserRightGapPositionNew/2-M_Compensation[j].Encoder)*(M_Compensation[j+1].RightTop-M_Compensation[j].RightTop))
						/(M_Compensation[j+1].Encoder-M_Compensation[j].Encoder))+M_Compensation[j].RightTop;
				RightBottomLinPositionNew:=(((UserRightGapPositionNew/2-M_Compensation[j].Encoder)*(M_Compensation[j+1].RightBottom-M_Compensation[j].RightBottom))
						/(M_Compensation[j+1].Encoder-M_Compensation[j].Encoder))+M_Compensation[j].RightBottom;
				M_CompensationNumber:=j;
				InitCompensationDatasDone:=TRUE;
			ELSIF j=18 AND UserRightGapPositionNew/2=M_Compensation[i].Encoder THEN		(*Gap=14µÄÌØÊâÇé¿ö*)
				(**)
				RightTopLinPositionNew:=M_Compensation[i].RightTop;
				RightBottomLinPositionNew:=M_Compensation[i].RightBottom;
				M_CompensationNumber:=j;
				InitCompensationDatasDone:=TRUE;
			ELSE
				RightTopLinPositionNew:=UserGapPositionNew/2;
				RightBottomLinPositionNew:=UserGapPositionNew/2;
				M_CompensationNumber:=j;
				InitCompensationDatasDone:=TRUE;
			END_IF
		END_IF
	END_FOR
	//
	//2.不论taper还是非taper模式，左轴gap都有左轴发推算，右轴gap由右轴反推算。taper为右gap-左gap
	//
	//左轴显示位置反结算
	FOR k:= 1 TO 17 DO
			IF Pos_LeftTopLin<M_Compensation[k+1].LeftTop AND Pos_LeftTopLin>=M_Compensation[k].LeftTop THEN
				UserGapPositionDisplay_FromLeftTop:=2*(((Pos_LeftTopLin-M_Compensation[k].LeftTop)*(M_Compensation[k+1].Encoder-M_Compensation[k].Encoder))
											/(M_Compensation[k+1].LeftTop-M_Compensation[k].LeftTop)+M_Compensation[k].Encoder);
				UserGapPositionDisplay_FromLeftBottom:=2*(((Pos_LeftBottomLin-M_Compensation[k].LeftBottom)*(M_Compensation[k+1].Encoder-M_Compensation[k].Encoder))
											/(M_Compensation[k+1].LeftBottom-M_Compensation[k].LeftBottom)+M_Compensation[k].Encoder);
				UserGapPositionDisplay:=DINT_TO_LREAL(LREAL_TO_DINT(((UserGapPositionDisplay_FromLeftTop+UserGapPositionDisplay_FromLeftBottom)/2)*100000))/100000;
			END_IF
	END_FOR
	//右轴显示位置反结算
	FOR m:= 1 TO 17 DO
			IF Pos_RightTopLin<M_Compensation[m+1].RightTop AND Pos_RightTopLin>=M_Compensation[m].RightTop THEN
				UserRightGapPositionDisplay_FromRightTop:=2*(((Pos_RightTopLin-M_Compensation[m].RightTop)*(M_Compensation[m+1].Encoder-M_Compensation[m].Encoder))
											/(M_Compensation[m+1].RightTop-M_Compensation[m].RightTop)+M_Compensation[m].Encoder);
				UserRightGapPositionDisplay_FromRightBottom:=2*(((Pos_RightBottomLin-M_Compensation[m].RightBottom)*(M_Compensation[m+1].Encoder-M_Compensation[m].Encoder))
											/(M_Compensation[m+1].RightBottom-M_Compensation[m].RightBottom)+M_Compensation[m].Encoder);
				UserRightGapPositionDisplay:=(UserRightGapPositionDisplay_FromRightTop+UserRightGapPositionDisplay_FromRightBottom)/2;
			END_IF
	END_FOR
	IF TaperOrNot OR (Global_ChainProtection_MPS_Triggered OR Global_ChainProtection_EPS_Triggered)  THEN//安全联锁触发时，需要UserTaperPositionDisplay作为A_MonitoringAllAxis的保护
		UserTaperPositionDisplay:=DINT_TO_LREAL(LREAL_TO_DINT((UserRightGapPositionDisplay-UserGapPositionDisplay)*100000))/100000;
		UserTaperVelocityDisplay:=DINT_TO_LREAL(LREAL_TO_DINT((Velo_RightTopLin+Velo_RightBottomLin)/2*100000))/100000;
	END_IF
END_IF
(*速度可以不用解算，直接用即可*)
LeftTopLinVelocityDisplay:=Velo_LeftTopLin;
RightTopLinVelocityDisplay:=Velo_RightTopLin;
LeftBottomLinVelocityDisplay:=Velo_LeftBottomLin;
RightBottomLinVelocityDisplay:=Velo_RightBottomLin;
//Gap velocity
UserGapVelocityDisplay:=DINT_TO_LREAL(LREAL_TO_DINT(((LeftTopLinVelocityDisplay+RightTopLinVelocityDisplay+
	LeftBottomLinVelocityDisplay+RightBottomLinVelocityDisplay)/2)*100000))/100000;

	(*解算单轴位置后，核验并做保护*)
	IF ABS(LeftTopLinPositionNew-UserGapPositionNew/2)>Threshold_motorsTargetPosCalculate THEN
		ErrorID:=1601;
		Error:=TRUE;
		ErrorDescription:='LeftTop Threshold_motorsTargetPosCalculate';
		FB_PlcEmergencyStop();
	END_IF
	//注意右轴解算以UserRightGapPositionNew为基准，考虑到taper
	IF ABS(RightTopLinPositionNew-UserRightGapPositionNew/2)>Threshold_motorsTargetPosCalculate THEN
		ErrorID:=1602;
		Error:=TRUE;
		ErrorDescription:='RightTop Threshold_motorsTargetPosCalculate';
		FB_PlcEmergencyStop();
	END_IF
	IF ABS(LeftBottomLinPositionNew-UserGapPositionNew/2)>Threshold_motorsTargetPosCalculate THEN
		ErrorID:=1603;
		Error:=TRUE;
		ErrorDescription:='LeftBottom Threshold_motorsTargetPosCalculate';
		FB_PlcEmergencyStop();
	END_IF
	//注意右轴解算以UserRightGapPositionNew为基准，考虑到taper
	IF ABS(RightBottomLinPositionNew-UserRightGapPositionNew/2)>Threshold_motorsTargetPosCalculate THEN
		ErrorID:=1604;
		Error:=TRUE;
		ErrorDescription:='RightBottom Threshold_motorsTargetPosCalculate';
		FB_PlcEmergencyStop();
	END_IF
END_ACTION

ACTION A_MonitoringAllAxis:
(****************************************************************
NAME:			A_MonitoringAllAxis
DATA:			2018.1.9
VERSION:		1.0.0
DESCRIPTION:	
				Ã¿´ÎÑ­»·¾ùÖ´ÐÐÖáÎ»ÖÃºÍÖáÔË¶¯µÄ¼ì²é
				2.4Öá¹âÕ¤³ßÎ»ÖÃ¡¢ËÙ¶È¶Ô±È¼ì²é
HISTORY:
				2017.1.9		NEW

***************************************************************)

(*************************************************************************************2.4Öá¹âÕ¤³ßÎ»ÖÃ¡¢ËÙ¶È¶Ô±È¼ì²é**********************************************************************)
IF  st_Power<>0 THEN
CASE moni_State OF
(*Top Î»ÖÃºÍËÙ¶È±È¶Ô*)
0:
		//实际(*Position*)
		(*Top*)
		Diff_UserTopPos_actual:=ABS(Pos_leftTopLin-Pos_RightTopLin);
		(*Bottom*)
		Diff_UserBottomPos_actual:=ABS(Pos_LeftBottomLin-Pos_RightBottomLin);
		(*Left*)
		Diff_UserLeftPos_actual:=ABS(Pos_LeftTopLin-Pos_LeftBottomLin);
		(*Right*)
		Diff_UserRightPos_actual:=ABS(Pos_RightTopLin-Pos_RightBottomLin);
		(*Velocity*)
		(*Top*)
		Diff_UserTopVelo_actual:=ABS(Velo_leftTopLin-Velo_RightTopLin);
		(*Bottom*)
		Diff_UserBottomVelo_actual:=ABS(Velo_LeftBottomLin-Velo_RightBottomLin);
		(*Left*)
		Diff_UserLeftVelo_actual:=ABS(Velo_LeftTopLin-Velo_LeftBottomLin);
		(*Right*)
		Diff_UserRightVelo_actual:=ABS(Velo_RightTopLin-Velo_RightBottomLin);
		//阈值
		Threshold_UserTopPos_PLC:=Threshold_UserTopPos+UserTaperPositionDisplay;//Top位置误差=gap运动细微误差+目标taper位置
		Threshold_UserTopVelo_PLC:=Threshold_UserTopVelo+ABS(UserGapVelocityDisplay);//Top速度误差=gap运动细微误差+gap目标速度。因为可能出现一个轴运动完了，另一个轴还在运动的情况
		Threshold_UserBottomPos_PLC:=Threshold_UserBottomPos+UserTaperPositionDisplay;//Bottom同上
		Threshold_UserBottomVelo_PLC:=Threshold_UserBottomVelo+ABS(UserGapVelocityDisplay);//Bottom同上
		Threshold_UserLeftPos_PLC:=Threshold_UserLeftPos+UserTaperPositionDisplay;
		Threshold_UserLeftVelo_PLC:=Threshold_UserLeftVelo+ABS(UserGapVelocityDisplay);
		Threshold_UserRightPos_PLC:=Threshold_UserRightPos+UserTaperPositionDisplay;
		Threshold_UserRightVelo_PLC:=Threshold_UserRightVelo+ABS(UserGapVelocityDisplay);
		//比较
		IF Diff_UserTopPos_actual >Threshold_UserTopPos_PLC THEN
				Error:=TRUE;
				ErrorID:=601;
				ErrorDescription:='Diff_UserTopPos_actual >Threshold_UserTopPos_PLC';
				moni_State:=-100;
		ELSIF Diff_UserTopVelo_actual>Threshold_UserTopVelo_PLC  THEN
				Error:=TRUE;
				ErrorID:=602;
				ErrorDescription:='Diff_UserTopVelo_actual>Threshold_UserTopVelo_PLC';
				moni_State:=-100;
		(*Bottom Î»ÖÃºÍËÙ¶È±È¶Ô*)
		ELSIF Diff_UserBottomPos_actual>Threshold_UserBottomPos_PLC THEN
				Error:=TRUE;
				ErrorID:=603;
				ErrorDescription:='Diff_UserBottomPos_actual>Threshold_UserBottomPos_PLC';
				moni_State:=-100;
		ELSIF Diff_UserBottomVelo_actual>Threshold_UserBottomVelo_PLC  THEN
				Error:=TRUE;
				ErrorID:=604;
				ErrorDescription:='Diff_UserBottomVelo_actual>Threshold_UserBottomVelo_PLC';
				moni_State:=-100;
		(*Left Î»ÖÃºÍËÙ¶È±È¶Ô*)
		ELSIF Diff_UserLeftPos_actual>Threshold_UserLeftPos_PLC  THEN
				Error:=TRUE;
				ErrorID:=605;
				ErrorDescription:='Diff_UserLeftPos_actual>Threshold_UserLeftPos_PLC';
				moni_State:=-100;
		ELSIF  Diff_UserLeftVelo_actual>Threshold_UserLeftVelo_PLC THEN
				Error:=TRUE;
				ErrorID:=606;
				ErrorDescription:='Diff_UserLeftVelo_actual>Threshold_UserLeftVelo_PLC';
				moni_State:=-100;
		(*Right Î»ÖÃºÍËÙ¶È±È¶Ô*)
		ELSIF Diff_UserRightPos_actual>Threshold_UserRightPos_PLC  THEN
				Error:=TRUE;
				ErrorID:=607;
				ErrorDescription:='Diff_UserRightPos_actual>Threshold_UserRightPos_PLC';
				moni_State:=-100;
		ELSIF  Diff_UserRightVelo_actual>Threshold_UserRightVelo_PLC THEN
				Error:=TRUE;
				ErrorID:=608;
				ErrorDescription:='Diff_UserRightVelo_actual>Threshold_UserRightVelo_PLC';
				moni_State:=-100;
		END_IF
-100:
		btn_UserGapStop:=TRUE;
		FB_PlcEmergencyStop();
		Error:=TRUE;
		LED_Error:=TRUE;
END_CASE
END_IF
END_ACTION

ACTION A_OneKeyToMaxGap:
//0.上升沿触发
//1.判断电机是否在开启状态,没有就打开电源
//2.判断是否在Moving状态,若有就Stop
//3.将磁间隙打开到至最大阈值
//4.到位后给出反馈
OneKeyToMaxGap_RTRIG(CLK:=btn_OneKeyToMaxGap);
IF OneKeyToMaxGap_RTRIG.Q THEN
	OneKeyToMaxGap_Triggered:=TRUE;
	OneKeyToMaxGap_Done:=FALSE;
END_IF
IF OneKeyToMaxGap_Triggered THEN
	CASE OneKeyToMaxGap_State OF
		0://1.判断电机是否在开启状态,没有就打开电源
			IF st_Power=1 THEN
				OneKeyToMaxGap_State:=1;
			ELSE
				btn_PowerOn:=TRUE;
				IF btn_PowerOn THEN
					A_PowerOn();
				END_IF
			END_IF
		1://1.判断是否在谱学扫描模式，如果是，则切换回正常运动模式
			IF IsSSMotionMode THEN
				SS_Stop:=TRUE;
				IsSSMotionMode:=FALSE;
			END_IF
			OneKeyToMaxGap_State:=2;
		2://判断是否在taper，如果在taper,则判断是否在运动，如果是，则停止运动,0.5sh后，转入下一步
			IF TaperOrNot THEN
				IF moveStatusLeftTop OR moveStatusRightTop OR moveStatusLeftBottom OR moveStatusRightBottom THEN
					btn_UserGapStop:=TRUE;
				ELSE
					OneKeyToMaxGap_TON_Stop2Move_InTaperMode(PT:=T#0.5S);
					OneKeyToMaxGap_TON_Stop2Move_InTaperMode.IN:=TRUE;
					IF OneKeyToMaxGap_TON_Stop2Move_InTaperMode.Q THEN
						TaperOrNot:=FALSE;//关闭taper模式
						OneKeyToMaxGap_State:=3;
						OneKeyToMaxGap_TON_Stop2Move_InTaperMode.IN:=FALSE;
					END_IF
				END_IF
			ELSE
				OneKeyToMaxGap_State:=3;
			END_IF
		3://3.判断是否在Moving状态,若有就Stop.Taper模式已处理完，此处开始走正常GAP开合逻辑
			IF moveStatusLeftTop OR moveStatusRightTop OR moveStatusLeftBottom OR moveStatusRightBottom THEN
				btn_UserGapStop:=TRUE;
			ELSE
				OneKeyToMaxGap_TON_Stop2Move(PT:=T#0.5S);
				OneKeyToMaxGap_TON_Stop2Move.IN:=TRUE;
				IF OneKeyToMaxGap_TON_Stop2Move.Q THEN
					OneKeyToMaxGap_State:=4;
					OneKeyToMaxGap_TON_Stop2Move.IN:=FALSE;
				END_IF
			END_IF
		4://4.将磁间隙打开到至最大阈值
			OneKeyToMaxGap_TON(PT:=INT_TO_TIME(LREAL_TO_INT(max_UserGapPositionNew+30))*1000);
			OneKeyToMaxGap_TON.IN:=TRUE;
			OneKeyToMaxGap_TON_Power2Move(PT:=T#0.1S);
			OneKeyToMaxGap_TON_Power2Move.IN:=TRUE;
			UserGapPositionNew:=max_UserGapPositionNew;
			UserGapVelocityNew:=1;
			btn_UserGapMove:=TRUE;
			IF OneKeyToMaxGap_TON_Power2Move.Q THEN
				OneKeyToMaxGap_TON_Power2Move.IN:=FALSE;
				IF FB_MOVE.BCGapDone THEN
					OneKeyToMaxGap_State:=88;
				END_IF
			END_IF
			IF OneKeyToMaxGap_TON.Q THEN//如果150s后，还没有运动到指定gap，则报错
				OneKeyToMaxGap_TON.IN:=FALSE;
				OneKeyToMaxGap_State:=-100;
			END_IF
		88://6.到位后给出反馈
			OneKeyToMaxGap_Done:=TRUE;	
			Error:=FALSE;
			ErrorID:=0;
			ErrorDescription:='';
			btn_OneKeyToMaxGap:=FALSE;
			OneKeyToMaxGap_Triggered:=FALSE;
			OneKeyToMaxGap_State:=0;
				
		-100:
			OneKeyToMaxGap_Done:=FALSE;
			Error:=TRUE;
			ErrorID:=1705;
			ErrorDescription:='OneKeyToMaxGap Fail';
			btn_OneKeyToMaxGap:=FALSE;
			OneKeyToMaxGap_Triggered:=FALSE;
			OneKeyToMaxGap_State:=0;
	END_CASE
END_IF
END_ACTION

ACTION A_PhaseLowerMotion:
IF btn_UserPhaseLowerMove THEN
	IF NOT inRange_UserPhaseLowerPositionNew THEN
		btn_UserPhaseLowerStop:=TRUE;
		btn_UserPhaseLowerMove:=FALSE;
		Error:=TRUE;
		ErrorId:=812;
		ErrorDescription:='target PhaseLower position out of range,please check';
		RETURN;
	ELSE
		btn_UserPhaseLowerStop:=FALSE;
		Error:=FALSE;
		ErrorId:=0;
		ErrorDescription:='';	
	END_IF
	IF NOT inRange_UserPhaseLowerVelocityNew THEN
		btn_UserPhaseLowerStop:=TRUE;
		btn_UserPhaseLowerMove:=FALSE;
		Error:=TRUE;
		ErrorId:=813;
		ErrorDescription:='target PhaseLower velocity out of range,please check';
		RETURN;
	ELSE
		btn_UserPhaseLowerStop:=FALSE;
		Error:=FALSE;
		ErrorId:=0;
		ErrorDescription:='';
	END_IF
END_IF

(*改变Phase前，先检查Gap，Gap必须处于阈值之上（基本在最大间隙），才能改变Phase*)
IF GapPhase_ChainProtection_On AND UserGapPositionDisplay-GapPhase_ChainProtection_MaxGapValue<-0.01 AND btn_UserPhaseLowerMove THEN
		btn_UserPhaseLowerStop:=TRUE;
		btn_UserPhaseLowerMove:=FALSE;
		Error:=TRUE;
		ErrorId:=814;
		ErrorDescription:='Please Move Gap to MaxGapValue first before move Phase';
		RETURN;
END_IF

(*Move*)
IF InitPowerDone THEN
	(*
	零位特殊走法入口。

	触发条件：
	1. 用户按下 PhaseLower Move；
	2. 当前没有执行过本次零位预走；
	3. 当前没有正在执行零位预走；
	4. 原 m/n 状态机都在空闲状态；
	5. 当前位置在零附近。

	重要说明：
	这里不提前判断正向/负向是否要走回程差。
	零位预走完成后，会重新进入原来的 m/n 判断。
	因此目标为负方向，例如 -10mm 时，流程是：
	0附近 -> 以慢速到 -ZeroBoundary -> 再进入原 n_state 回程差逻辑。
	*)
	IF btn_UserPhaseLowerMove
		AND EnableZeroPre_PhaseLower
		AND NOT ZeroPreDone_PhaseLower
		AND NOT ZeroPreMoving_PhaseLower
		AND m_state_PhaseLower=0
		AND n_state_PhaseLower=0
		AND ABS(Pos_PhaseLowerLin)<=ZeroNearThreshold_PhaseLower THEN

		IF NOT st_Power THEN
			ErrorID:=1501;
			Error:=TRUE;
			ErrorDescription:='Plz PowerOn Frist';
			LED_Error:=TRUE;
			RETURN;
		ELSE
			ErrorID:=0;
			Error:=FALSE;
			ErrorDescription:='';
			LED_Error:=FALSE;
		END_IF

		(*锁存本次用户目标和速度，避免零位慢速段期间 HMI 输入变化影响本次运动。*)
		ZeroFinalTarget_PhaseLower:=UserPhaseLowerPositionNew;
		ZeroFinalVelocity_PhaseLower:=UserPhaseLowerVelocityNew;

		(*
		如果目标在 +/-ZeroBoundary_PhaseLower 内：
		直接以 ZeroSlowVelocity_PhaseLower 走到最终目标，本次运动结束。

		如果目标超过边界：
		先以 ZeroSlowVelocity_PhaseLower 走到 +ZeroBoundary 或 -ZeroBoundary。
		走完后再进入原 m/n 正常逻辑，保留回程差判断。
		*)
		IF ABS(ZeroFinalTarget_PhaseLower)<=ZeroBoundary_PhaseLower THEN
			ZeroPreTarget_PhaseLower:=ZeroFinalTarget_PhaseLower;
			ZeroDirectMove_PhaseLower:=TRUE;
		ELSE
			IF ZeroFinalTarget_PhaseLower>ZeroBoundary_PhaseLower THEN
				ZeroPreTarget_PhaseLower:=ZeroBoundary_PhaseLower;
			ELSE
				ZeroPreTarget_PhaseLower:=-ZeroBoundary_PhaseLower;
			END_IF
			ZeroDirectMove_PhaseLower:=FALSE;
		END_IF

		ZeroPreMoving_PhaseLower:=TRUE;
		z_state_PhaseLower:=10;
	END_IF

	IF ZeroPreMoving_PhaseLower THEN
		CASE z_state_PhaseLower OF
			10:
				(*
				零位预走发命令。
				这里的目标一定是：
				1. 边界内目标：最终目标；
				2. 边界外目标：+ZeroBoundary 或 -ZeroBoundary。
				速度固定使用 ZeroSlowVelocity_PhaseLower。
				*)
				FB_Move_PhaseLower.Mode:=4;						//1.gap;2.single;3.taper;4.debug;5.BCGap&UserMode
				FB_Move_PhaseLower.CoupleState:=st_Couple;			
				FB_Move_PhaseLower.PowerState:=st_Power;			
				FB_Move_PhaseLower.PhaseLowerPosition:=ZeroPreTarget_PhaseLower;
				FB_Move_PhaseLower.PhaseLowerVelocity:=ZeroSlowVelocity_PhaseLower;
				FB_Move_PhaseLower.PhaseLowerMove:=TRUE;
				btn_UserPhaseLowerMove:=FALSE;
				Led_Run:=TRUE;
				FB_Move_PhaseLower();
				z_state_PhaseLower:=11;

			11:
				(*等待零位预走到位。*)
				btn_UserPhaseLowerMove:=FALSE;
				FB_Move_PhaseLower();
				IF NOT FB_Move_PhaseLower.PhaseLowerDone THEN
					Led_Run:=TRUE;
					z_state_PhaseLower:=11;
				ELSE
					(*
					到位后先撤掉 Move 信号。
					下一拍再决定是结束，还是进入原 m/n 正常逻辑。
					这样和原 n_state 两段运动的处理方式一致：两段之间给 FB 一个 Move=FALSE 的间隔。
					*)
					FB_Move_PhaseLower.PhaseLowerMove:=FALSE;
					FB_Move_PhaseLower();
					z_state_PhaseLower:=12;
				END_IF

			12:
				(*
				零位预走完成后的分流。

				ZeroDirectMove_PhaseLower=TRUE：
					目标本来就在 +/-ZeroBoundary 内，慢速走到目标后本次运动直接结束。

				ZeroDirectMove_PhaseLower=FALSE：
					目标超过边界，只完成了“慢速离开零位”。
					此时设置 ZeroPreDone=TRUE，并重新置 btn_UserPhaseLowerMove=TRUE。
					下一扫描周期会跳过零位预走入口，进入原 m/n 正常逻辑。
				*)
				FB_Move_PhaseLower.PhaseLowerMove:=FALSE;
				FB_Move_PhaseLower.PhaseLowerReset:=FALSE;
				FB_Move_PhaseLower();

				IF ZeroDirectMove_PhaseLower THEN
					z_state_PhaseLower:=88;
				ELSE
					ZeroPreMoving_PhaseLower:=FALSE;
					ZeroPreDone_PhaseLower:=TRUE;
					btn_UserPhaseLowerMove:=TRUE;
					Led_Run:=FALSE;
					z_state_PhaseLower:=0;
				END_IF

			88:
				(*零位直达目标的收尾。*)
				btn_UserPhaseLowerMove:=FALSE;
				FB_Move_PhaseLower.PhaseLowerMove:=FALSE;
				FB_Move_PhaseLower.PhaseLowerReset:=FALSE;
				Led_Run:=FALSE;
				z_state_PhaseLower:=0;
				ZeroPreMoving_PhaseLower:=FALSE;
				ZeroPreDone_PhaseLower:=FALSE;
				ZeroDirectMove_PhaseLower:=FALSE;
		END_CASE

	ELSE
		(*
		原 m/n 正常逻辑。

		重要说明：
		如果刚执行完零位预走，ZeroPreDone_PhaseLower=TRUE，
		这里使用锁存的 ZeroFinalTarget/ZeroFinalVelocity。
		否则仍使用 HMI 当前给定的 UserPhaseLowerPositionNew/UserPhaseLowerVelocityNew。
		*)
		IF ZeroPreDone_PhaseLower THEN
			ActiveTarget_PhaseLower:=ZeroFinalTarget_PhaseLower;
			ActiveVelocity_PhaseLower:=ZeroFinalVelocity_PhaseLower;
		ELSE
			ActiveTarget_PhaseLower:=UserPhaseLowerPositionNew;
			ActiveVelocity_PhaseLower:=UserPhaseLowerVelocityNew;
		END_IF

		(*分别比较四轴目标位置与当前位置的差，如果目标位置比当前位置低，则需要运动到更低-回程差一半；再运动至最终目标位置*)
		//只在m=和n=0的时候判断，否则会出现一些BUG，比如往大间隙开时，运动到位后m不能回到0.
		IF m_state_PhaseLower=0 AND n_state_PhaseLower=0 THEN
			IF ActiveTarget_PhaseLower-Pos_PhaseLowerLin<-LEDriftErrorThreshold_PhaseLower THEN
					TargetPosLessThanCurrentPos_PhaseLower:=TRUE;
			ELSE
					TargetPosLessThanCurrentPos_PhaseLower:=FALSE;
			END_IF
		END_IF

		(*目标位置大于当前位置，直接走到目标位置，不需要先走到考虑回程误差的临时位置。*)
		IF NOT TargetPosLessThanCurrentPos_PhaseLower AND NOT HysteresisMoving_PhaseLower THEN
			CASE m_state_PhaseLower OF
				0:
					FB_Move_PhaseLower.Mode:=4;						//1.gap;2.single;3.taper;4.debug;5.BCGap&UserMode
					FB_Move_PhaseLower.CoupleState:=st_Couple;			
					FB_Move_PhaseLower.PowerState:=st_Power;	
					IF btn_UserPhaseLowerMove THEN						
						IF NOT st_Power THEN
							ErrorID:=1501;
							Error:=TRUE;
							ErrorDescription:='Plz PowerOn Frist';
							LED_Error:=TRUE;
							RETURN;
						ELSE
							ErrorID:=0;
							Error:=FALSE;
							ErrorDescription:='';
							LED_Error:=FALSE;
						END_IF
						//目标速度位置赋值
						FB_Move_PhaseLower.PhaseLowerPosition:=ActiveTarget_PhaseLower;
						FB_Move_PhaseLower.PhaseLowerVelocity:=ActiveVelocity_PhaseLower;		
						//Move
						FB_Move_PhaseLower.PhaseLowerMove:=TRUE;
						m_state_PhaseLower:=1;
						FB_Move_PhaseLower();
					END_IF

				1:
					btn_UserPhaseLowerMove:=FALSE;
					FB_Move_PhaseLower();
					IF NOT FB_Move_PhaseLower.PhaseLowerDone THEN			(*运动未完成，循环等待*)
						Led_Run:=TRUE;
						m_state_PhaseLower:=1;
					ELSE									(*运动完成，进入收尾*)
						m_state_PhaseLower:=88;
					END_IF

				88:
					btn_UserPhaseLowerMove:=FALSE;					(*状态恢复*)
					Led_Run:=FALSE;
					m_state_PhaseLower:=0;
					ZeroPreDone_PhaseLower:=FALSE;
					ZeroPreMoving_PhaseLower:=FALSE;
					ZeroDirectMove_PhaseLower:=FALSE;
					z_state_PhaseLower:=0;
			END_CASE

		(*目标位置小于当前位置，保留原回程差逻辑：先走到临时位置，再走到最终位置。*)
		ELSE
			CASE n_state_PhaseLower OF
				0:
					FB_Move_PhaseLower.Mode:=4;						//1.gap;2.single;3.taper;4.debug;5.BCGap&UserMode;5:userMode_2
					FB_Move_PhaseLower.CoupleState:=st_Couple;			
					FB_Move_PhaseLower.PowerState:=st_Power;			
					IF btn_UserPhaseLowerMove THEN
						IF NOT st_Power THEN
							ErrorID:=1501;
							Error:=TRUE;
							ErrorDescription:='Plz PowerOn Frist';
							LED_Error:=TRUE;
							RETURN;
						ELSE
							ErrorID:=0;
							Error:=FALSE;
							ErrorDescription:='';
							LED_Error:=FALSE;
						END_IF

						IF TargetPosLessThanCurrentPos_PhaseLower THEN			
							FB_Move_PhaseLower.PhaseLowerPosition:=ActiveTarget_PhaseLower-HysteresisError_PhaseLower;
						ELSE
							FB_Move_PhaseLower.PhaseLowerPosition:=ActiveTarget_PhaseLower;	
						END_IF				

						(*
						锁定最终目标。
						原程序这里锁 UserPhaseLowerPositionNewTemp，是为了避免运动过程中目标输入变化。
						这里改为锁 ActiveTarget_PhaseLower：
						- 普通运动时 ActiveTarget=UserPhaseLowerPositionNew；
						- 零位预走后 ActiveTarget=ZeroFinalTarget_PhaseLower。
						*)
						UserPhaseLowerPositionNewTemp:=ActiveTarget_PhaseLower;
						FB_Move_PhaseLower.PhaseLowerVelocity:=ActiveVelocity_PhaseLower;
						
						FB_Move_PhaseLower.PhaseLowerMove:=TRUE;
						FB_Move_PhaseLower();
						HysteresisMoving_PhaseLower:=TRUE;
						n_state_PhaseLower:=1;
					END_IF

				1:
					btn_UserPhaseLowerMove:=FALSE;
					FB_Move_PhaseLower();
					IF NOT FB_Move_PhaseLower.PhaseLowerDone THEN			(*还未运动到临时位置，运动过程中*)
						Led_Run:=TRUE;
						n_state_PhaseLower:=1;
					ELSE									
						n_state_PhaseLower:=2;							(*转到下一步，运动到最终位置*)
						FB_Move_PhaseLower.PhaseLowerMove:=FALSE;
					END_IF

				2:
					FB_Move_PhaseLower.PhaseLowerReset:=FALSE;
					FB_Move_PhaseLower.Mode:=4;						//1.gap;2.single;3.taper;4.debug;5.BCGap&UserMode
					FB_Move_PhaseLower.CoupleState:=st_Couple;			
					FB_Move_PhaseLower.PowerState:=st_Power;			
					FB_Move_PhaseLower.PhaseLowerMove:=TRUE;
					//直接走到最终目标。最终目标已在 n_state=0 中锁存到 UserPhaseLowerPositionNewTemp。
					FB_Move_PhaseLower.PhaseLowerPosition:=UserPhaseLowerPositionNewTemp;	
					FB_Move_PhaseLower.PhaseLowerVelocity:=ActiveVelocity_PhaseLower;
					FB_Move_PhaseLower();							
					n_state_PhaseLower:=3;

				3:
					FB_Move_PhaseLower();
					IF NOT FB_Move_PhaseLower.PhaseLowerDone THEN			(*还未运动到最终位置，运动过程中*)
						Led_Run:=TRUE;
						n_state_PhaseLower:=3;
					ELSE									
						n_state_PhaseLower:=88;							(*运动到了最终位置*)
					END_IF

				88:
					btn_UserPhaseLowerMove:=FALSE;					
					Led_Run:=FALSE;
					n_state_PhaseLower:=0;
					HysteresisMoving_PhaseLower:=FALSE;
					ZeroPreDone_PhaseLower:=FALSE;
					ZeroPreMoving_PhaseLower:=FALSE;
					ZeroDirectMove_PhaseLower:=FALSE;
					z_state_PhaseLower:=0;
			END_CASE
		END_IF
	END_IF
END_IF

IF btn_UserPhaseLowerStop THEN
	FB_Move_PhaseLower.PhaseLowerReset:=TRUE;							(*给运动FB停止/复位信号，使FB_Move状态恢复*)
	FB_Move_PhaseLower();											(*启动FB_Move*)
	btn_UserPhaseLowerMove:=FALSE;
	m_state_PhaseLower:=0;	
	n_state_PhaseLower:=0;

	(*Stop 时必须同时清零位预走相关状态，避免停止后残留在特殊流程中。*)
	z_state_PhaseLower:=0;
	ZeroPreMoving_PhaseLower:=FALSE;
	ZeroPreDone_PhaseLower:=FALSE;
	ZeroDirectMove_PhaseLower:=FALSE;

	CASE s_state_PhaseLower OF
			0:
				FB_Stop_PhaseLower.Mode:=4;							(*1:gap模式; 2:单梁模式; 3:taper模式; 4:Debug模式; 5:BCGap模式*)
				FB_Stop_PhaseLower.CoupleState:=st_Couple;			(*耦合状态输入*)
				FB_Stop_PhaseLower.PowerState:=st_Power;				(*电源状态输入*)
				FB_Stop_PhaseLower.PhaseLowerStop:=TRUE;				(*Execute TRUE*)
				FB_Stop_PhaseLower();								(*启动FB*)
				s_state_PhaseLower:=1;
			1:
				FB_Stop_PhaseLower();
				IF NOT FB_Stop_PhaseLower.PhaseLowerDone THEN			(*停止未完成，循环*)
					s_state_PhaseLower:=1;
				ELSE									(*停止完成，下一步*)
					s_state_PhaseLower:=88;
				END_IF
			88:
				btn_UserPhaseLowerStop:=FALSE;						(*恢复状态*)
				FB_Move_PhaseLower.PhaseLowerReset:=FALSE;				(*运行FB*)
				s_state_PhaseLower:=0;
		END_CASE
END_IF

(*触发限位开关后，相当于点击了Stop按钮*)
FTrig_ReachLS_PhaseLower(CLK:=LS_PhaseLower_Entrance AND LS_PhaseLower_Exit);
IF FTrig_ReachLS_PhaseLower.Q THEN
	btn_UserPhaseLowerStop:=TRUE;
END_IF
END_ACTION

ACTION A_PhaseLowerMotion_1:
(*输入保护*)
IF btn_UserPhaseLowerMove THEN
	IF NOT inRange_UserPhaseLowerPositionNew THEN
		btn_UserPhaseLowerStop:=TRUE;
		btn_UserPhaseLowerMove:=FALSE;
		Error:=TRUE;
		ErrorId:=812;
		ErrorDescription:='target PhaseLower position out of range,please check';
		RETURN;
	ELSE
		btn_UserPhaseLowerStop:=FALSE;
		Error:=FALSE;
		ErrorId:=0;
		ErrorDescription:='';	
	END_IF
	IF NOT inRange_UserPhaseLowerVelocityNew THEN
		btn_UserPhaseLowerStop:=TRUE;
		btn_UserPhaseLowerMove:=FALSE;
		Error:=TRUE;
		ErrorId:=813;
		ErrorDescription:='target PhaseLower velocity out of range,please check';
		RETURN;
	ELSE
		btn_UserPhaseLowerStop:=FALSE;
		Error:=FALSE;
		ErrorId:=0;
		ErrorDescription:='';
	END_IF
END_IF
(*改变Phase前，先检查Gap，Gap必须处于阈值之上（基本在最大间隙），才能改变Pase*)
IF GapPhase_ChainProtection_On AND UserGapPositionDisplay-GapPhase_ChainProtection_MaxGapValue<-0.01 AND btn_UserPhaseLowerMove THEN
		btn_UserPhaseLowerStop:=TRUE;
		btn_UserPhaseLowerMove:=FALSE;
		Error:=TRUE;
		ErrorId:=814;
		ErrorDescription:='Please Move Gap to MaxGapValue first before move Phase';
		RETURN;
END_IF

(*分别比较四轴目标位置与当前位置的差，如果目标位置比当前位置低，则需要运动到更低-回程差一半；再运动至最终目标位置*)
//只在m=和n=0的时候判断，否则会出现一些BUG，比如往大间隙开时，运动到位后m不能回到0.
IF m_state_PhaseLower=0 AND n_state_PhaseLower=0 THEN
	IF UserPhaseLowerPositionNew-Pos_PhaseLowerLin<-LEDriftErrorThreshold_PhaseLower THEN
			TargetPosLessThanCurrentPos_PhaseLower:=TRUE;
	ELSE
			TargetPosLessThanCurrentPos_PhaseLower:=FALSE;
	END_IF
END_IF

(*Move*)
IF InitPowerDone THEN
		(*目标位置都大于当前位置，直接走到目标位置即可，不需要先走到考虑回城误差的临时位置*)
		IF NOT TargetPosLessThanCurrentPos_PhaseLower AND NOT HysteresisMoving_PhaseLower THEN
			CASE m_state_PhaseLower OF
				0:
					FB_Move_PhaseLower.Mode:=4;						//1.gap;2.single;3.taper;4.debug;5.BCGap&UserMode
					FB_Move_PhaseLower.CoupleState:=st_Couple;			
					FB_Move_PhaseLower.PowerState:=st_Power;							
					FB_Move_PhaseLower.PhaseLowerPosition:=UserPhaseLowerPositionNew;
					FB_Move_PhaseLower.PhaseLowerVelocity:=UserPhaseLowerVelocityNew;		
					IF btn_UserPhaseLowerMove THEN
						FB_Move_PhaseLower.PhaseLowerMove:=TRUE;
						m_state_PhaseLower:=1;
						FB_Move_PhaseLower();
					END_IF
				1:
					btn_UserPhaseLowerMove:=FALSE;
					FB_Move_PhaseLower();
					IF NOT FB_Move_PhaseLower.PhaseLowerDone THEN			(*ÔË¶¯Î´Íê³É£¬Ñ­»·*)
						Led_Run:=TRUE;
						m_state_PhaseLower:=1;
					ELSE									(*ÔË¶¯Íê³É£¬ÏÂÒ»²½*)
						m_state_PhaseLower:=88;
					END_IF
				88:
					btn_UserPhaseLowerMove:=FALSE;					(*×´Ì¬»Ö¸´*)
					Led_Run:=FALSE;
					m_state_PhaseLower:=0;
			END_CASE
		(*四轴有目标位置小于当前位置，先走到临时位置，再走到目标位置*)
		ELSE
			CASE n_state_PhaseLower OF
				0:
					FB_Move_PhaseLower.Mode:=4;						//1.gap;2.single;3.taper;4.debug;5.BCGap&UserMode;5:userMode_2
					FB_Move_PhaseLower.CoupleState:=st_Couple;			
					FB_Move_PhaseLower.PowerState:=st_Power;			
					
					//
					IF TargetPosLessThanCurrentPos_PhaseLower THEN			
						FB_Move_PhaseLower.PhaseLowerPosition:=UserPhaseLowerPositionNew-HysteresisError_PhaseLower;
					ELSE
						FB_Move_PhaseLower.PhaseLowerPosition:=UserPhaseLowerPositionNew;	
					END_IF				
					//
					FB_Move_PhaseLower.PhaseLowerVelocity:=UserPhaseLowerVelocityNew;
						
					IF btn_UserPhaseLowerMove THEN							
						n_state_PhaseLower:=1;
						FB_Move_PhaseLower.PhaseLowerMove:=TRUE;
						FB_Move_PhaseLower();
						HysteresisMoving_PhaseLower:=TRUE;
					END_IF
				1:
					btn_UserPhaseLowerMove:=FALSE;
					FB_Move_PhaseLower();
					IF NOT FB_Move_PhaseLower.PhaseLowerDone THEN			(*还未运动到位置,运动过程中*)
						Led_Run:=TRUE;
						n_state_PhaseLower:=1;
					ELSE									
						n_state_PhaseLower:=2;							(*转到下一步，运动到最终位置*)
						FB_Move_PhaseLower.PhaseLowerMove:=FALSE;
						//Led_Run:=FALSE;
					END_IF
				2:
					FB_Move_PhaseLower.PhaseLowerReset:=FALSE;
					FB_Move_PhaseLower.Mode:=4;						//1.gap;2.single;3.taper;4.debug;5.BCGap&UserMode
					FB_Move_PhaseLower.CoupleState:=st_Couple;			
					FB_Move_PhaseLower.PowerState:=st_Power;			
					FB_Move_PhaseLower.PhaseLowerMove:=TRUE;
					//直接走到目标位置，已经走到位置的，可以继续下命令，只不过它不在走了而已
					FB_Move_PhaseLower.PhaseLowerPosition:=UserPhaseLowerPositionNew;	
					FB_Move_PhaseLower.PhaseLowerVelocity:=UserPhaseLowerVelocityNew;
					FB_Move_PhaseLower();							
					n_state_PhaseLower:=3;
				3:
					FB_Move_PhaseLower();
					IF NOT FB_Move_PhaseLower.PhaseLowerDone THEN			(*还未运动到位置,运动过程中*)
						Led_Run:=TRUE;
						n_state_PhaseLower:=3;
					ELSE									
						n_state_PhaseLower:=88;							(*运动到了最终位置*)
					END_IF
				88:
					btn_UserPhaseLowerMove:=FALSE;					
					Led_Run:=FALSE;
					n_state_PhaseLower:=0;
					HysteresisMoving_PhaseLower:=FALSE;
			END_CASE
		END_IF
	//END_IF
END_IF

IF btn_UserPhaseLowerStop THEN
	FB_Move_PhaseLower.PhaseLowerReset:=TRUE;							(*¸øÔË¶¯FB¸øÍ£Ö¹ÐÅºÅ£¬Ê¹FB_Move×´Ì¬»Ö¸´*)
	FB_Move_PhaseLower();											(*Æô¶¯FB_Move*)
	btn_UserPhaseLowerMove:=FALSE;								(*btn_GapMove:=FALSE*)
	m_state_PhaseLower:=0;	
	n_state_PhaseLower:=0;										(*m_state:=0;*)
	CASE s_state_PhaseLower OF
			0:
				FB_Stop_PhaseLower.Mode:=4;							(*1£ºgapÄ£Ê½£»2£ºµ¥ÁºÄ£Ê½£»3£ºtaperÄ£Ê½£»4£ºDebugÄ£Ê½£»5£ºBCGapÄ£Ê½*)
				FB_Stop_PhaseLower.CoupleState:=st_Couple;			(*ñîºÏ×´Ì¬ÊäÈë*)
				FB_Stop_PhaseLower.PowerState:=st_Power;				(*µçÔ´×´Ì¬ÊäÈë*)
				FB_Stop_PhaseLower.PhaseLowerStop:=TRUE;				(*Execute TRUE*)
				FB_Stop_PhaseLower();								(*Æô¶¯FB*)
				s_state_PhaseLower:=1;
			1:
				FB_Stop_PhaseLower();
				IF NOT FB_Stop_PhaseLower.PhaseLowerDone THEN			(*Í£Ö¹Î´Íê³É£¬Ñ­»·*)
					s_state_PhaseLower:=1;
				ELSE									(*Í£Ö¹Íê³É£¬ÏÂÒ»²½*)
					s_state_PhaseLower:=88;
				END_IF
			88:
				btn_UserPhaseLowerStop:=FALSE;						(*»Ö¸´×´Ì¬*)
				FB_Move_PhaseLower.PhaseLowerReset:=FALSE;				(*ÔËÐÐFB*)
				s_state_PhaseLower:=0;
		END_CASE
END_IF

(*触发限位开关后，相当于点击了Stop按钮*)
FTrig_ReachLS_PhaseLower(CLK:=LS_PhaseLower_Entrance AND LS_PhaseLower_Exit);
IF FTrig_ReachLS_PhaseLower.Q THEN
	btn_UserPhaseLowerStop:=TRUE;
END_IF
END_ACTION

ACTION A_PhaseUpperMotion:
(*输入保护*)
IF btn_UserPhaseUpperMove THEN
	IF NOT inRange_UserPhaseUpperPositionNew THEN
		btn_UserPhaseUpperStop:=TRUE;
		btn_UserPhaseUpperMove:=FALSE;
		Error:=TRUE;
		ErrorId:=809;
		ErrorDescription:='target PhaseUpper position out of range,please check';
		RETURN;
	ELSE
		btn_UserPhaseUpperStop:=FALSE;
		Error:=FALSE;
		ErrorId:=0;
		ErrorDescription:='';	
	END_IF
	IF NOT inRange_UserPhaseUpperVelocityNew THEN
		btn_UserPhaseUpperStop:=TRUE;
		btn_UserPhaseUpperMove:=FALSE;
		Error:=TRUE;
		ErrorId:=810;
		ErrorDescription:='target PhaseUpper velocity out of range,please check';
		RETURN;
	ELSE
		btn_UserPhaseUpperStop:=FALSE;
		Error:=FALSE;
		ErrorId:=0;
		ErrorDescription:='';
	END_IF
END_IF

(*改变Phase前，先检查Gap，Gap必须处于阈值之上（基本在最大间隙），才能改变Phase*)
IF GapPhase_ChainProtection_On AND UserGapPositionDisplay-GapPhase_ChainProtection_MaxGapValue<-0.01 AND btn_UserPhaseUpperMove THEN
		btn_UserPhaseUpperStop:=TRUE;
		btn_UserPhaseUpperMove:=FALSE;
		Error:=TRUE;
		ErrorId:=811;
		ErrorDescription:='Please Move Gap to MaxGapValue first before move Phase';
		RETURN;
END_IF

(*Move*)
IF InitPowerDone THEN
	(*
	零位特殊走法入口。

	触发条件：
	1. 用户按下 PhaseUpper Move；
	2. 当前没有执行过本次零位预走；
	3. 当前没有正在执行零位预走；
	4. 原 m/n 状态机都在空闲状态；
	5. 当前位置在零附近。

	重要说明：
	这里不提前判断正向/负向是否要走回程差。
	零位预走完成后，会重新进入原来的 m/n 判断。
	因此目标为负方向，例如 -10mm 时，流程是：
	0附近 -> 以慢速到 -ZeroBoundary -> 再进入原 n_state 回程差逻辑。
	*)
	IF btn_UserPhaseUpperMove
		AND EnableZeroPre_PhaseUpper
		AND NOT ZeroPreDone_PhaseUpper
		AND NOT ZeroPreMoving_PhaseUpper
		AND m_state_PhaseUpper=0
		AND n_state_PhaseUpper=0
		AND ABS(Pos_PhaseUpperLin)<=ZeroNearThreshold_PhaseUpper THEN

		IF NOT st_Power THEN
			ErrorID:=1501;
			Error:=TRUE;
			ErrorDescription:='Plz PowerOn Frist';
			LED_Error:=TRUE;
			RETURN;
		ELSE
			ErrorID:=0;
			Error:=FALSE;
			ErrorDescription:='';
			LED_Error:=FALSE;
		END_IF

		(*锁存本次用户目标和速度，避免零位慢速段期间 HMI 输入变化影响本次运动。*)
		ZeroFinalTarget_PhaseUpper:=UserPhaseUpperPositionNew;
		ZeroFinalVelocity_PhaseUpper:=UserPhaseUpperVelocityNew;

		(*
		如果目标在 +/-ZeroBoundary_PhaseUpper 内：
		直接以 ZeroSlowVelocity_PhaseUpper 走到最终目标，本次运动结束。
		如果目标超过边界：
		先以 ZeroSlowVelocity_PhaseUpper 走到 +ZeroBoundary 或 -ZeroBoundary。
		走完后再进入原 m/n 正常逻辑，保留回程差判断。
		*)
		IF ABS(ZeroFinalTarget_PhaseUpper)<=ZeroBoundary_PhaseUpper THEN
			ZeroPreTarget_PhaseUpper:=ZeroFinalTarget_PhaseUpper;
			ZeroDirectMove_PhaseUpper:=TRUE;
		ELSE
			IF ZeroFinalTarget_PhaseUpper>ZeroBoundary_PhaseUpper THEN
				ZeroPreTarget_PhaseUpper:=ZeroBoundary_PhaseUpper;
			ELSE
				ZeroPreTarget_PhaseUpper:=-ZeroBoundary_PhaseUpper;
			END_IF
			ZeroDirectMove_PhaseUpper:=FALSE;
		END_IF

		ZeroPreMoving_PhaseUpper:=TRUE;
		z_state_PhaseUpper:=10;
	END_IF

	IF ZeroPreMoving_PhaseUpper THEN
		CASE z_state_PhaseUpper OF
			10:
				(*
				零位预走发命令。
				这里的目标一定是：
				1. 边界内目标：最终目标；
				2. 边界外目标：+ZeroBoundary 或 -ZeroBoundary。
				速度固定使用 ZeroSlowVelocity_PhaseUpper。
				*)
				FB_Move_PhaseUpper.Mode:=4;						//1.gap;2.single;3.taper;4.debug;5.BCGap&UserMode
				FB_Move_PhaseUpper.CoupleState:=st_Couple;			
				FB_Move_PhaseUpper.PowerState:=st_Power;			
				FB_Move_PhaseUpper.PhaseUpperPosition:=ZeroPreTarget_PhaseUpper;
				FB_Move_PhaseUpper.PhaseUpperVelocity:=ZeroSlowVelocity_PhaseUpper;
				FB_Move_PhaseUpper.PhaseUpperMove:=TRUE;
				btn_UserPhaseUpperMove:=FALSE;
				Led_Run:=TRUE;
				FB_Move_PhaseUpper();
				z_state_PhaseUpper:=11;

			11:
				(*等待零位预走到位。*)
				btn_UserPhaseUpperMove:=FALSE;
				FB_Move_PhaseUpper();
				IF NOT FB_Move_PhaseUpper.PhaseUpperDone THEN
					Led_Run:=TRUE;
					z_state_PhaseUpper:=11;
				ELSE
					(*
					到位后先撤掉 Move 信号。
					下一拍再决定是结束，还是进入原 m/n 正常逻辑。
					这样和原 n_state 两段运动的处理方式一致：两段之间给 FB 一个 Move=FALSE 的间隔。
					*)
					FB_Move_PhaseUpper.PhaseUpperMove:=FALSE;
					FB_Move_PhaseUpper();
					z_state_PhaseUpper:=12;
				END_IF

			12:
				(*
				零位预走完成后的分流。

				ZeroDirectMove_PhaseUpper=TRUE：
					目标本来就在 +/-ZeroBoundary 内，慢速走到目标后本次运动直接结束。
				ZeroDirectMove_PhaseUpper=FALSE：
					目标超过边界，只完成了“慢速离开零位”。
					此时设置 ZeroPreDone=TRUE，并重新置 btn_UserPhaseUpperMove=TRUE。
					下一扫描周期会跳过零位预走入口，进入原 m/n 正常逻辑。
				*)
				FB_Move_PhaseUpper.PhaseUpperMove:=FALSE;
				FB_Move_PhaseUpper.PhaseUpperReset:=FALSE;
				FB_Move_PhaseUpper();

				IF ZeroDirectMove_PhaseUpper THEN
					z_state_PhaseUpper:=88;
				ELSE
					ZeroPreMoving_PhaseUpper:=FALSE;
					ZeroPreDone_PhaseUpper:=TRUE;
					btn_UserPhaseUpperMove:=TRUE;
					Led_Run:=FALSE;
					z_state_PhaseUpper:=0;
				END_IF

			88:
				(*零位直达目标的收尾。*)
				btn_UserPhaseUpperMove:=FALSE;
				FB_Move_PhaseUpper.PhaseUpperMove:=FALSE;
				FB_Move_PhaseUpper.PhaseUpperReset:=FALSE;
				Led_Run:=FALSE;
				z_state_PhaseUpper:=0;
				ZeroPreMoving_PhaseUpper:=FALSE;
				ZeroPreDone_PhaseUpper:=FALSE;
				ZeroDirectMove_PhaseUpper:=FALSE;
		END_CASE

	ELSE
		(*
		原 m/n 正常逻辑。
		重要说明：
		如果刚执行完零位预走，ZeroPreDone_PhaseUpper=TRUE，
		这里使用锁存的 ZeroFinalTarget/ZeroFinalVelocity。
		否则仍使用 HMI 当前给定的 UserPhaseUpperPositionNew/UserPhaseUpperVelocityNew。
		*)
		IF ZeroPreDone_PhaseUpper THEN
			ActiveTarget_PhaseUpper:=ZeroFinalTarget_PhaseUpper;
			ActiveVelocity_PhaseUpper:=ZeroFinalVelocity_PhaseUpper;
		ELSE
			ActiveTarget_PhaseUpper:=UserPhaseUpperPositionNew;
			ActiveVelocity_PhaseUpper:=UserPhaseUpperVelocityNew;
		END_IF

		(*分别比较四轴目标位置与当前位置的差，如果目标位置比当前位置低，则需要运动到更低-回程差一半；再运动至最终目标位置*)
		//只在m=和n=0的时候判断，否则会出现一些BUG，比如往大间隙开时，运动到位后m不能回到0.
		IF m_state_PhaseUpper=0 AND n_state_PhaseUpper=0 THEN
			IF ActiveTarget_PhaseUpper-Pos_PhaseUpperLin<-LEDriftErrorThreshold_PhaseUpper THEN
					TargetPosLessThanCurrentPos_PhaseUpper:=TRUE;
			ELSE
					TargetPosLessThanCurrentPos_PhaseUpper:=FALSE;
			END_IF
		END_IF

		(*目标位置大于当前位置，直接走到目标位置，不需要先走到考虑回程误差的临时位置。*)
		IF NOT TargetPosLessThanCurrentPos_PhaseUpper AND NOT HysteresisMoving_PhaseUpper THEN
			CASE m_state_PhaseUpper OF
				0:
					FB_Move_PhaseUpper.Mode:=4;						//1.gap;2.single;3.taper;4.debug;5.BCGap&UserMode
					FB_Move_PhaseUpper.CoupleState:=st_Couple;			
					FB_Move_PhaseUpper.PowerState:=st_Power;	
					IF btn_UserPhaseUpperMove THEN						
						IF NOT st_Power THEN
							ErrorID:=1501;
							Error:=TRUE;
							ErrorDescription:='Plz PowerOn Frist';
							LED_Error:=TRUE;
							RETURN;
						ELSE
							ErrorID:=0;
							Error:=FALSE;
							ErrorDescription:='';
							LED_Error:=FALSE;
						END_IF
						//目标速度位置赋值
						FB_Move_PhaseUpper.PhaseUpperPosition:=ActiveTarget_PhaseUpper;
						FB_Move_PhaseUpper.PhaseUpperVelocity:=ActiveVelocity_PhaseUpper;		
						//Move
						FB_Move_PhaseUpper.PhaseUpperMove:=TRUE;
						m_state_PhaseUpper:=1;
						FB_Move_PhaseUpper();
					END_IF

				1:
					btn_UserPhaseUpperMove:=FALSE;
					FB_Move_PhaseUpper();
					IF NOT FB_Move_PhaseUpper.PhaseUpperDone THEN			(*运动未完成，循环等待*)
						Led_Run:=TRUE;
						m_state_PhaseUpper:=1;
					ELSE									(*运动完成，进入收尾*)
						m_state_PhaseUpper:=88;
					END_IF

				88:
					btn_UserPhaseUpperMove:=FALSE;					(*状态恢复*)
					Led_Run:=FALSE;
					m_state_PhaseUpper:=0;
					ZeroPreDone_PhaseUpper:=FALSE;
					ZeroPreMoving_PhaseUpper:=FALSE;
					ZeroDirectMove_PhaseUpper:=FALSE;
					z_state_PhaseUpper:=0;
			END_CASE

		(*目标位置小于当前位置，保留原回程差逻辑：先走到临时位置，再走到最终位置。*)
		ELSE
			CASE n_state_PhaseUpper OF
				0:
					FB_Move_PhaseUpper.Mode:=4;						//1.gap;2.single;3.taper;4.debug;5.BCGap&UserMode;5:userMode_2
					FB_Move_PhaseUpper.CoupleState:=st_Couple;			
					FB_Move_PhaseUpper.PowerState:=st_Power;			
					IF btn_UserPhaseUpperMove THEN
						IF NOT st_Power THEN
							ErrorID:=1501;
							Error:=TRUE;
							ErrorDescription:='Plz PowerOn Frist';
							LED_Error:=TRUE;
							RETURN;
						ELSE
							ErrorID:=0;
							Error:=FALSE;
							ErrorDescription:='';
							LED_Error:=FALSE;
						END_IF

						IF TargetPosLessThanCurrentPos_PhaseUpper THEN			
							FB_Move_PhaseUpper.PhaseUpperPosition:=ActiveTarget_PhaseUpper-HysteresisError_PhaseUpper;
						ELSE
							FB_Move_PhaseUpper.PhaseUpperPosition:=ActiveTarget_PhaseUpper;	
						END_IF				

						(*
						锁定最终目标。
						原程序这里锁 UserPhaseUpperPositionNewTemp，是为了避免运动过程中目标输入变化。
						这里改为锁 ActiveTarget_PhaseUpper：
						- 普通运动时 ActiveTarget=UserPhaseUpperPositionNew；
						- 零位预走后 ActiveTarget=ZeroFinalTarget_PhaseUpper。
						*)
						UserPhaseUpperPositionNewTemp:=ActiveTarget_PhaseUpper;
						FB_Move_PhaseUpper.PhaseUpperVelocity:=ActiveVelocity_PhaseUpper;
						
						FB_Move_PhaseUpper.PhaseUpperMove:=TRUE;
						FB_Move_PhaseUpper();
						HysteresisMoving_PhaseUpper:=TRUE;
						n_state_PhaseUpper:=1;
					END_IF

				1:
					btn_UserPhaseUpperMove:=FALSE;
					FB_Move_PhaseUpper();
					IF NOT FB_Move_PhaseUpper.PhaseUpperDone THEN			(*还未运动到临时位置，运动过程中*)
						Led_Run:=TRUE;
						n_state_PhaseUpper:=1;
					ELSE									
						n_state_PhaseUpper:=2;							(*转到下一步，运动到最终位置*)
						FB_Move_PhaseUpper.PhaseUpperMove:=FALSE;
					END_IF

				2:
					FB_Move_PhaseUpper.PhaseUpperReset:=FALSE;
					FB_Move_PhaseUpper.Mode:=4;						//1.gap;2.single;3.taper;4.debug;5.BCGap&UserMode
					FB_Move_PhaseUpper.CoupleState:=st_Couple;			
					FB_Move_PhaseUpper.PowerState:=st_Power;			
					FB_Move_PhaseUpper.PhaseUpperMove:=TRUE;
					//直接走到最终目标。最终目标已在 n_state=0 中锁存到 UserPhaseUpperPositionNewTemp。
					FB_Move_PhaseUpper.PhaseUpperPosition:=UserPhaseUpperPositionNewTemp;	
					FB_Move_PhaseUpper.PhaseUpperVelocity:=ActiveVelocity_PhaseUpper;
					FB_Move_PhaseUpper();							
					n_state_PhaseUpper:=3;

				3:
					FB_Move_PhaseUpper();
					IF NOT FB_Move_PhaseUpper.PhaseUpperDone THEN			(*还未运动到最终位置，运动过程中*)
						Led_Run:=TRUE;
						n_state_PhaseUpper:=3;
					ELSE									
						n_state_PhaseUpper:=88;							(*运动到了最终位置*)
					END_IF

				88:
					btn_UserPhaseUpperMove:=FALSE;					
					Led_Run:=FALSE;
					n_state_PhaseUpper:=0;
					HysteresisMoving_PhaseUpper:=FALSE;
					ZeroPreDone_PhaseUpper:=FALSE;
					ZeroPreMoving_PhaseUpper:=FALSE;
					ZeroDirectMove_PhaseUpper:=FALSE;
					z_state_PhaseUpper:=0;
			END_CASE
		END_IF
	END_IF
END_IF

IF btn_UserPhaseUpperStop THEN
	FB_Move_PhaseUpper.PhaseUpperReset:=TRUE;							(*给运动FB停止/复位信号，使FB_Move状态恢复*)
	FB_Move_PhaseUpper();											(*启动FB_Move*)
	btn_UserPhaseUpperMove:=FALSE;
	m_state_PhaseUpper:=0;	
	n_state_PhaseUpper:=0;

	(*Stop 时必须同时清零位预走相关状态，避免停止后残留在特殊流程中。*)
	z_state_PhaseUpper:=0;
	ZeroPreMoving_PhaseUpper:=FALSE;
	ZeroPreDone_PhaseUpper:=FALSE;
	ZeroDirectMove_PhaseUpper:=FALSE;

	CASE s_state_PhaseUpper OF
			0:
				FB_Stop_PhaseUpper.Mode:=4;							(*1:gap模式; 2:单梁模式; 3:taper模式; 4:Debug模式; 5:BCGap模式*)
				FB_Stop_PhaseUpper.CoupleState:=st_Couple;			(*耦合状态输入*)
				FB_Stop_PhaseUpper.PowerState:=st_Power;				(*电源状态输入*)
				FB_Stop_PhaseUpper.PhaseUpperStop:=TRUE;				(*Execute TRUE*)
				FB_Stop_PhaseUpper();								(*启动FB*)
				s_state_PhaseUpper:=1;
			1:
				FB_Stop_PhaseUpper();
				IF NOT FB_Stop_PhaseUpper.PhaseUpperDone THEN			(*停止未完成，循环*)
					s_state_PhaseUpper:=1;
				ELSE									(*停止完成，下一步*)
					s_state_PhaseUpper:=88;
				END_IF
			88:
				btn_UserPhaseUpperStop:=FALSE;						(*恢复状态*)
				FB_Move_PhaseUpper.PhaseUpperReset:=FALSE;				(*运行FB*)
				s_state_PhaseUpper:=0;
		END_CASE
END_IF

(*触发限位开关后，相当于点击了Stop按钮*)
FTrig_ReachLS_PhaseUpper(CLK:=LS_PhaseUpper_Entrance AND LS_PhaseUpper_Exit);
IF FTrig_ReachLS_PhaseUpper.Q THEN
	btn_UserPhaseUpperStop:=TRUE;
END_IF
END_ACTION

ACTION A_PhaseUpperMotion_1:
(*输入保护*)
IF btn_UserPhaseUpperMove THEN
	IF NOT inRange_UserPhaseUpperPositionNew THEN
		btn_UserPhaseUpperStop:=TRUE;
		btn_UserPhaseUpperMove:=FALSE;
		Error:=TRUE;
		ErrorId:=809;
		ErrorDescription:='target PhaseUpper position out of range,please check';
		RETURN;
	ELSE
		btn_UserPhaseUpperStop:=FALSE;
		Error:=FALSE;
		ErrorId:=0;
		ErrorDescription:='';	
	END_IF
	IF NOT inRange_UserPhaseUpperVelocityNew THEN
		btn_UserPhaseUpperStop:=TRUE;
		btn_UserPhaseUpperMove:=FALSE;
		Error:=TRUE;
		ErrorId:=810;
		ErrorDescription:='target PhaseUpper velocity out of range,please check';
		RETURN;
	ELSE
		btn_UserPhaseUpperStop:=FALSE;
		Error:=FALSE;
		ErrorId:=0;
		ErrorDescription:='';
	END_IF
END_IF
(*改变Phase前，先检查Gap，Gap必须处于阈值之上（基本在最大间隙），才能改变Pase*)
IF GapPhase_ChainProtection_On AND UserGapPositionDisplay-GapPhase_ChainProtection_MaxGapValue<-0.01 AND btn_UserPhaseUpperMove THEN
		btn_UserPhaseUpperStop:=TRUE;
		btn_UserPhaseUpperMove:=FALSE;
		Error:=TRUE;
		ErrorId:=811;
		ErrorDescription:='Please Move Gap to MaxGapValue first before move Phase';
		RETURN;
END_IF
(*分别比较四轴目标位置与当前位置的差，如果目标位置比当前位置低，则需要运动到更低-回程差一半；再运动至最终目标位置*)
//只在m=和n=0的时候判断，否则会出现一些BUG，比如往大间隙开时，运动到位后m不能回到0.
IF m_state_PhaseUpper=0 AND n_state_PhaseUpper=0 THEN
	IF UserPhaseUpperPositionNew-Pos_PhaseUpperLin<-LEDriftErrorThreshold_PhaseUpper THEN
			TargetPosLessThanCurrentPos_PhaseUpper:=TRUE;
	ELSE
			TargetPosLessThanCurrentPos_PhaseUpper:=FALSE;
	END_IF
END_IF

(*Move*)
IF InitPowerDone THEN
		(*目标位置都大于当前位置，直接走到目标位置即可，不需要先走到考虑回城误差的临时位置*)
		IF NOT TargetPosLessThanCurrentPos_PhaseUpper AND NOT HysteresisMoving_PhaseUpper THEN
			CASE m_state_PhaseUpper OF
				0:
					FB_Move_PhaseUpper.Mode:=4;						//1.gap;2.single;3.taper;4.debug;5.BCGap&UserMode
					FB_Move_PhaseUpper.CoupleState:=st_Couple;			
					FB_Move_PhaseUpper.PowerState:=st_Power;	
					IF btn_UserPhaseUpperMove THEN						
						IF NOT st_Power THEN
							ErrorID:=1501;
							Error:=TRUE;
							ErrorDescription:='Plz PowerOn Frist';
							LED_Error:=TRUE;
							//btn_UserGapMove:=FALSE;
							RETURN;
						ELSE
							ErrorID:=0;
							Error:=FALSE;
							ErrorDescription:='';
							LED_Error:=FALSE;
							//btn_UserGapMove:=TRUE;
						END_IF
						//目标速度位置赋值
						FB_Move_PhaseUpper.PhaseUpperPosition:=UserPhaseUpperPositionNew;
						FB_Move_PhaseUpper.PhaseUpperVelocity:=UserPhaseUpperVelocityNew;		
						//Move
						FB_Move_PhaseUpper.PhaseUpperMove:=TRUE;
						m_state_PhaseUpper:=1;
						FB_Move_PhaseUpper();
					END_IF
				1:
					btn_UserPhaseUpperMove:=FALSE;
					FB_Move_PhaseUpper();
					IF NOT FB_Move_PhaseUpper.PhaseUpperDone THEN			(*ÔË¶¯Î´Íê³É£¬Ñ­»·*)
						Led_Run:=TRUE;
						m_state_PhaseUpper:=1;
					ELSE									(*ÔË¶¯Íê³É£¬ÏÂÒ»²½*)
						m_state_PhaseUpper:=88;
					END_IF
				88:
					btn_UserPhaseUpperMove:=FALSE;					(*×´Ì¬»Ö¸´*)
					Led_Run:=FALSE;
					m_state_PhaseUpper:=0;
			END_CASE
		(*四轴有目标位置小于当前位置，先走到临时位置，再走到目标位置*)
		ELSE
			CASE n_state_PhaseUpper OF
				0:
					FB_Move_PhaseUpper.Mode:=4;						//1.gap;2.single;3.taper;4.debug;5.BCGap&UserMode;5:userMode_2
					FB_Move_PhaseUpper.CoupleState:=st_Couple;			
					FB_Move_PhaseUpper.PowerState:=st_Power;			
					//
					IF btn_UserPhaseUpperMove THEN
						IF NOT st_Power THEN
							ErrorID:=1501;
							Error:=TRUE;
							ErrorDescription:='Plz PowerOn Frist';
							LED_Error:=TRUE;
							//btn_UserGapMove:=FALSE;
							RETURN;
						ELSE
							ErrorID:=0;
							Error:=FALSE;
							ErrorDescription:='';
							LED_Error:=FALSE;
							//btn_UserGapMove:=TRUE;	
						END_IF
						IF TargetPosLessThanCurrentPos_PhaseUpper THEN			
							FB_Move_PhaseUpper.PhaseUpperPosition:=UserPhaseUpperPositionNew-HysteresisError_PhaseUpper;
						ELSE
							FB_Move_PhaseUpper.PhaseUpperPosition:=UserPhaseUpperPositionNew;	
						END_IF				
						//	close gap情况下，加入了PositionNewTemp。//
						//如果在往小间隙运行过程中，改变了目标gap，会在第到达第一次目标位置后，继续向第二
						//次输入的目标运动，而不会回到第一次的目标位置。用temp锁定目标位置
						UserPhaseUpperPositionNewTemp:=UserPhaseUpperPositionNew;
						FB_Move_PhaseUpper.PhaseUpperVelocity:=UserPhaseUpperVelocityNew;
						
						FB_Move_PhaseUpper.PhaseUpperMove:=TRUE;
						FB_Move_PhaseUpper();
						HysteresisMoving_PhaseUpper:=TRUE;
						n_state_PhaseUpper:=1;
					END_IF
				1:
					btn_UserPhaseUpperMove:=FALSE;
					FB_Move_PhaseUpper();
					IF NOT FB_Move_PhaseUpper.PhaseUpperDone THEN			(*还未运动到位置,运动过程中*)
						Led_Run:=TRUE;
						n_state_PhaseUpper:=1;
					ELSE									
						n_state_PhaseUpper:=2;							(*转到下一步，运动到最终位置*)
						FB_Move_PhaseUpper.PhaseUpperMove:=FALSE;
						//Led_Run:=FALSE;
					END_IF
				2:
					FB_Move_PhaseUpper.PhaseUpperReset:=FALSE;
					FB_Move_PhaseUpper.Mode:=4;						//1.gap;2.single;3.taper;4.debug;5.BCGap&UserMode
					FB_Move_PhaseUpper.CoupleState:=st_Couple;			
					FB_Move_PhaseUpper.PowerState:=st_Power;			
					FB_Move_PhaseUpper.PhaseUpperMove:=TRUE;
					//直接走到目标位置，已经走到位置的，可以继续下命令，只不过它不在走了而已
					FB_Move_PhaseUpper.PhaseUpperPosition:=UserPhaseUpperPositionNewTemp;	
					FB_Move_PhaseUpper.PhaseUpperVelocity:=UserPhaseUpperVelocityNew;
					FB_Move_PhaseUpper();							
					n_state_PhaseUpper:=3;
				3:
					FB_Move_PhaseUpper();
					IF NOT FB_Move_PhaseUpper.PhaseUpperDone THEN			(*还未运动到位置,运动过程中*)
						Led_Run:=TRUE;
						n_state_PhaseUpper:=3;
					ELSE									
						n_state_PhaseUpper:=88;							(*运动到了最终位置*)
					END_IF
				88:
					btn_UserPhaseUpperMove:=FALSE;					
					Led_Run:=FALSE;
					n_state_PhaseUpper:=0;
					HysteresisMoving_PhaseUpper:=FALSE;
			END_CASE
		END_IF
	//END_IF
END_IF

IF btn_UserPhaseUpperStop THEN
	FB_Move_PhaseUpper.PhaseUpperReset:=TRUE;							(*¸øÔË¶¯FB¸øÍ£Ö¹ÐÅºÅ£¬Ê¹FB_Move×´Ì¬»Ö¸´*)
	FB_Move_PhaseUpper();											(*Æô¶¯FB_Move*)
	btn_UserPhaseUpperMove:=FALSE;								(*btn_GapMove:=FALSE*)
	m_state_PhaseUpper:=0;	
	n_state_PhaseUpper:=0;										(*m_state:=0;*)
	CASE s_state_PhaseUpper OF
			0:
				FB_Stop_PhaseUpper.Mode:=4;							(*1£ºgapÄ£Ê½£»2£ºµ¥ÁºÄ£Ê½£»3£ºtaperÄ£Ê½£»4£ºDebugÄ£Ê½£»5£ºBCGapÄ£Ê½*)
				FB_Stop_PhaseUpper.CoupleState:=st_Couple;			(*ñîºÏ×´Ì¬ÊäÈë*)
				FB_Stop_PhaseUpper.PowerState:=st_Power;				(*µçÔ´×´Ì¬ÊäÈë*)
				FB_Stop_PhaseUpper.PhaseUpperStop:=TRUE;				(*Execute TRUE*)
				FB_Stop_PhaseUpper();								(*Æô¶¯FB*)
				s_state_PhaseUpper:=1;
			1:
				FB_Stop_PhaseUpper();
				IF NOT FB_Stop_PhaseUpper.PhaseUpperDone THEN			(*Í£Ö¹Î´Íê³É£¬Ñ­»·*)
					s_state_PhaseUpper:=1;
				ELSE									(*Í£Ö¹Íê³É£¬ÏÂÒ»²½*)
					s_state_PhaseUpper:=88;
				END_IF
			88:
				btn_UserPhaseUpperStop:=FALSE;						(*»Ö¸´×´Ì¬*)
				FB_Move_PhaseUpper.PhaseUpperReset:=FALSE;				(*ÔËÐÐFB*)
				s_state_PhaseUpper:=0;
		END_CASE
END_IF

(*触发限位开关后，相当于点击了Stop按钮*)
FTrig_ReachLS_PhaseUpper(CLK:=LS_PhaseUpper_Entrance AND LS_PhaseUpper_Exit);
IF FTrig_ReachLS_PhaseUpper.Q THEN
	btn_UserPhaseUpperStop:=TRUE;
END_IF
END_ACTION

ACTION A_PowerOff:
CASE d_state OF
		0:(*PowerOff*)
			FB_Power(Off:=TRUE);
				d_state:=1;
		1:
			IF NOT FB_power.OffStatus THEN
				d_state:=1;
			ELSE
				d_state:=88;
			END_IF
		88:(*ResetAllState*)
			btn_PowerOn:=FALSE;
			btn_UserGapMove:=FALSE;
			btn_UserGapStop:=FALSE;
			LeftTopLinMoveIndicator:=0;
			RightTopLinMoveIndicator:=0;
			LeftBottomLinMoveIndicator:=0;
			RightBottomLinMoveIndicator:=0;
			fb_ton1.IN:=FALSE;
			fb_ton2.IN:=FALSE;
			fb_ton3.IN:=FALSE;
			State:=0;
			Busy:=FALSE;
			InitPowerDone:=FALSE;
			InitCompensationDatasDone:=FALSE;
			Error:=FALSE;
			ErrorID:=0;
			m_state:=0;
			n_state:=0;
			s_state:=0;
			btn_PowerOff:=FALSE;
			d_state:=0;
			Led_Run:=FALSE;
			Led_Error:=FALSE;
			moni_State:=0;
			i:=0;
END_CASE
END_ACTION

ACTION A_PowerOn:
(****************************************************************
NAME:			A_PowerOn
DATA:			2018.1.9
VERSION:		1.0.0
DESCRIPTION:	
				ÉÏµãÃüÁîºó£¬Ë³ÐòÖ´ÐÐ£º
				1.FB_PowerOn
				·µ»ØÖ´ÐÐÊÇ·ñ³É¹¦
HISTORY:
				2019.1.9		NEW

***************************************************************)
fb_ton3(PT:=t#0.5s);
CASE State OF
	0:	(*FB_Power_On*)
		FB_Power(On:=TRUE);
		fb_ton3.IN:=TRUE;
		State:=1;
	1:	(*wait*)
		FB_power();
		IF NOT FB_power.OnStatus THEN		(*FB_Power_OnÃ»ÓÐÖ´ÐÐÍê£¬wait£¬³¬Ê±FB Error*)
			IF NOT fb_ton3.Q THEN
				State:=1;
			ELSE
				ErrorID:=1;
				State:=99;
			END_IF
		ELSE
			State:=88;
		END_IF
	88:	(*All Done*)
		btn_PowerOn:=FALSE;
		State:=0;
		Error:=FALSE;
		ErrorID:=0;
		Busy:=FALSE;
		InitPowerDone:=TRUE;
		FB_power.On:=FALSE;
		fb_ton3.IN:=FALSE;
		LED_Error:=FALSE;
	99:
		Error:=TRUE;
		//ErrorID:=701;
		//ErrorDescription:='power on error';		
		btn_PowerOn:=FALSE;
		State:=99;
		Busy:=FALSE;
		InitPowerDone:=FALSE;
		fb_ton3.IN:=FALSE;
		LED_Error:=TRUE;
END_CASE
END_ACTION

ACTION A_RegularMotion:
(*如果该ID没有taper需求，则TaperFunctionSolidOn=FALSE，则判定taperOrNot为false*)
IF NOT TaperFunctionSolidOn THEN
	TaperOrNot:=FALSE;
END_IF

(*分别比较四轴目标位置与当前位置的差，如果目标位置比当前位置低，则需要运动到更低-回程差一半；再运动至最终目标位置*)
//只在m=和n=0的时候判断，否则会出现一些BUG，比如往大间隙开时，运动到位后m不能回到0.
IF m_state=0 AND n_state=0 THEN
		TargetPosLessThanCurrentPos:=FALSE;
	IF LeftTopLinPositionNew-Pos_LeftTopLin<-LEDriftErrorThreshold THEN
			TargetPosLessThanCurrentPos:=TRUE;
			TargetLTPosLessThanCurrentLTPos:=TRUE;
	ELSE
				TargetLTPosLessThanCurrentLTPos:=FALSE;
	END_IF
	IF RightTopLinPositionNew-Pos_RightTopLin<-LEDriftErrorThreshold THEN
			TargetPosLessThanCurrentPos:=TRUE;
			TargetRTPosLessThanCurrentRTPos:=TRUE;
	ELSE
			TargetRTPosLessThanCurrentRTPos:=FALSE;
	END_IF
	IF LeftBottomLinPositionNew-Pos_LeftBottomLin<-LEDriftErrorThreshold THEN
			TargetPosLessThanCurrentPos:=TRUE;
			TargetLBPosLessThanCurrentLBPos:=TRUE;
	ELSE
			TargetLBPosLessThanCurrentLBPos:=FALSE;
	END_IF
	IF RightBottomLinPositionNew-Pos_RightBottomLin<-LEDriftErrorThreshold THEN
			TargetPosLessThanCurrentPos:=TRUE;
			TargetRBPosLessThanCurrentRBPos:=TRUE;
	ELSE
			TargetRBPosLessThanCurrentRBPos:=FALSE;
	END_IF
END_IF

(*Move*)
IF InitCompensationDatasDone THEN
		(*四轴目标位置都大于当前位置，直接走到目标位置即可，不需要先走到考虑回城误差的临时位置*)
		IF NOT TargetPosLessThanCurrentPos AND NOT HysteresisMoving THEN
			CASE m_state OF
				0:
					FB_Move.Mode:=5;						//1.gap;2.single;3.taper;4.debug;5.BCGap&UserMode
					FB_Move.CoupleState:=st_Couple;			
					FB_Move.PowerState:=st_Power;						
			
					IF btn_UserGapMove THEN					
						moveStatusGap:=TRUE;
						FB_Move.BCGapReset:=TRUE;
						IF NOT st_Power THEN
							ErrorID:=1501;
							Error:=TRUE;
							ErrorDescription:='Plz PowerOn Frist';
							LED_Error:=TRUE;
							//btn_UserGapMove:=FALSE;
							RETURN;
						ELSE
							ErrorID:=0;
							Error:=FALSE;
							ErrorDescription:='';
							LED_Error:=FALSE;
							//btn_UserGapMove:=TRUE;
						END_IF
						//目标速度位置赋值
						FB_Move.BCLeftTopPosition:=LeftTopLinPositionNew;
						FB_Move.BCRightTopPosition:=RightTopLinPositionNew;
						FB_Move.BCLeftBottomPosition:=LeftBottomLinPositionNew;
						FB_Move.BCRightBottomPosition:=RightBottomLinPositionNew;
						IF NOT TaperOrNot THEN
							FB_Move.BCLeftTopVelocity:=UserGapVelocityNew/2;
							FB_Move.BCRightTopVelocity:=UserGapVelocityNew/2;
							FB_Move.BCLeftBottomVelocity:=UserGapVelocityNew/2;
							FB_Move.BCRightBottomVelocity:=UserGapVelocityNew/2;
						ELSE
							FB_Move.BCLeftTopVelocity:=UserTaperVelocityNew;
							FB_Move.BCRightTopVelocity:=UserTaperVelocityNew;
							FB_Move.BCLeftBottomVelocity:=UserTaperVelocityNew;
							FB_Move.BCRightBottomVelocity:=UserTaperVelocityNew;
						END_IF
						m_state:=1;
						FB_Move();
					END_IF
				1:
					FB_Move.BCGapMove:=TRUE;
					btn_UserGapMove:=FALSE;
					FB_Move();
					IF NOT FB_Move.BCGapDone THEN			(*ÔË¶¯Î´Íê³É£¬Ñ­»·*)
						Led_Run:=TRUE;
						m_state:=1;
					ELSE									(*ÔË¶¯Íê³É£¬ÏÂÒ»²½*)
						m_state:=88;
					END_IF
				88:
					moveStatusGap:=FALSE;
					btn_UserGapMove:=FALSE;					(*×´Ì¬»Ö¸´*)
					Led_Run:=FALSE;
					m_state:=0;
			END_CASE
		(*四轴有目标位置小于当前位置，先走到临时位置，再走到目标位置*)
		ELSE
			CASE n_state OF
				0:
					FB_Move.Mode:=5;						//1.gap;2.single;3.taper;4.debug;5.BCGap&UserMode;5:userMode_2
					FB_Move.CoupleState:=st_Couple;			
					FB_Move.PowerState:=st_Power;			
					IF btn_UserGapMove THEN	
						FB_Move.BCGapReset:=TRUE;					
						moveStatusGap:=TRUE;
						IF NOT st_Power THEN
							ErrorID:=1501;
							Error:=TRUE;
							ErrorDescription:='Plz PowerOn Frist';
							LED_Error:=TRUE;
							//btn_UserGapMove:=FALSE;
							RETURN;
						ELSE
							ErrorID:=0;
							Error:=FALSE;
							ErrorDescription:='';
							LED_Error:=FALSE;
							//btn_UserGapMove:=TRUE;
						END_IF						
						//
						IF TargetLTPosLessThanCurrentLTPos THEN			
							FB_Move.BCLeftTopPosition:=LeftTopLinPositionNew-HysteresisError/2;
						ELSE
							FB_Move.BCLeftTopPosition:=LeftTopLinPositionNew;	
						END_IF
						//
						IF TargetRTPosLessThanCurrentRTPos THEN 
							FB_Move.BCRightTopPosition:=RightTopLinPositionNew-HysteresisError/2;
						ELSE					
							FB_Move.BCRightTopPosition:=RightTopLinPositionNew;
						END_IF
						//
						IF TargetLBPosLessThanCurrentLBPos THEN
							FB_Move.BCLeftBottomPosition:=LeftBottomLinPositionNew-HysteresisError/2;
						ELSE
							FB_Move.BCLeftBottomPosition:=LeftBottomLinPositionNew;
						END_IF
						//
						IF TargetRBPosLessThanCurrentRBPos THEN
							FB_Move.BCRightBottomPosition:=RightBottomLinPositionNew-HysteresisError/2;
						ELSE
							FB_Move.BCRightBottomPosition:=RightBottomLinPositionNew;
						END_IF	
						//	close gap情况下，加入了LeftTopLinPositionNewTemp。//
						//如果在往小间隙运行过程中，改变了目标gap，会在第到达第一次目标位置后，继续向第二
						//次输入的目标运动，而不会回到第一次的目标位置。用temp锁定目标位置
						LeftTopLinPositionNewTemp:=LeftTopLinPositionNew;
						RightTopLinPositionNewTemp:=RightTopLinPositionNew;
						LeftBottomLinPositionNewTemp:=LeftBottomLinPositionNew;
						RightBottomLinPositionNewTemp:=RightBottomLinPositionNew;
			
						//
						IF NOT TaperOrNot THEN
							FB_Move.BCLeftTopVelocity:=UserGapVelocityNew/2;
							FB_Move.BCRightTopVelocity:=UserGapVelocityNew/2;
							FB_Move.BCLeftBottomVelocity:=UserGapVelocityNew/2;
							FB_Move.BCRightBottomVelocity:=UserGapVelocityNew/2;
							IF UserGapVelocityNew >1 THEN								  
								ErrorID:=1502;
								Error:=TRUE;
								ErrorDescription:='UserGapVelocityNew must<=1';
								LED_Error:=TRUE;
								btn_UserGapMove:=FALSE;
								RETURN;
							ELSE
								ErrorID:=0;
								Error:=FALSE;
								ErrorDescription:='';
								LED_Error:=FALSE;	
							END_IF									
						ELSE
							FB_Move.BCLeftTopVelocity:=UserTaperVelocityNew;
							FB_Move.BCRightTopVelocity:=UserTaperVelocityNew;
							FB_Move.BCLeftBottomVelocity:=UserTaperVelocityNew;
							FB_Move.BCRightBottomVelocity:=UserTaperVelocityNew;
						END_IF	

						FB_Move();
						HysteresisMoving:=TRUE;		
						n_state:=1;	
					END_IF
				1:
					btn_UserGapMove:=FALSE;	
					FB_Move.BCGapMove:=TRUE;
					FB_Move();
					IF NOT FB_Move.BCGapDone THEN			(*还未运动到位置,运动过程中*)
						Led_Run:=TRUE;
						n_state:=1;
					ELSE									
						n_state:=2;							(*转到下一步，运动到最终位置*)
						FB_Move.BCGapMove:=FALSE;
						//Led_Run:=FALSE;
					END_IF
				2:
					FB_Move.BCGapReset:=FALSE;
					FB_Move.Mode:=5;						//1.gap;2.single;3.taper;4.debug;5.BCGap&UserMode
					FB_Move.CoupleState:=st_Couple;			
					FB_Move.PowerState:=st_Power;			
					FB_Move.BCGapMove:=TRUE;
					//直接走到目标位置，已经走到位置的，可以继续下命令，只不过它不在走了而已
					FB_Move.BCLeftTopPosition:=LeftTopLinPositionNewTemp;	
					FB_Move.BCRightTopPosition:=RightTopLinPositionNewTemp;
					FB_Move.BCLeftBottomPosition:=LeftBottomLinPositionNewTemp;
					FB_Move.BCRightBottomPosition:=RightBottomLinPositionNewTemp;
					//
					IF NOT TaperOrNot THEN
						FB_Move.BCLeftTopVelocity:=UserGapVelocityNew/2;
						FB_Move.BCRightTopVelocity:=UserGapVelocityNew/2;
						FB_Move.BCLeftBottomVelocity:=UserGapVelocityNew/2;
						FB_Move.BCRightBottomVelocity:=UserGapVelocityNew/2;
					ELSE
						FB_Move.BCLeftTopVelocity:=UserTaperVelocityNew;
						FB_Move.BCRightTopVelocity:=UserTaperVelocityNew;
						FB_Move.BCLeftBottomVelocity:=UserTaperVelocityNew;
						FB_Move.BCRightBottomVelocity:=UserTaperVelocityNew;
					END_IF
					FB_Move();							
					n_state:=3;
				3:
					FB_Move();
					IF NOT FB_Move.BCGapDone THEN			(*还未运动到位置,运动过程中*)
						Led_Run:=TRUE;
						n_state:=3;
					ELSE									
						n_state:=88;							(*运动到了最终位置*)
					END_IF
					(*
					IF NOT Unreach_LS_Bottom THEN
						n_state:=88;							(*在运动过程中如果碰到下限位，则也转到下一步，运动到最终位置*)
						FB_Move.BCGapMove_2:=FALSE;
					END_IF
					*)
				88:				
					moveStatusGap:=FALSE;
					btn_UserGapMove:=FALSE;					
					Led_Run:=FALSE;
					n_state:=0;
					HysteresisMoving:=FALSE;
			END_CASE
		END_IF
	//
	//FB_Move.BCLeftTopPosition等四轴位置监控
	//
END_IF

//
//STOP
//
CASE s_state OF
	0:
		IF btn_UserGapStop OR btn_Reset THEN					
			moveStatusGap:=FALSE;
			m_state:=0;	
			n_state:=0;	
			HysteresisMoving:=FALSE;
					
			FB_Stop.Mode:=5;	
			FB_Stop.CoupleState:=st_Couple;	
			FB_Stop.PowerState:=st_Power;
			FB_Stop.BCGapStop:=TRUE;
			FB_Stop();	
			s_state:=1;
		END_IF
	1:
		btn_UserGapStop:=FALSE;	
		FB_Stop();
		IF NOT FB_Stop.BCGapDone THEN
			s_state:=1;
		ELSE
			s_state:=88;
		END_IF
	88:
		FB_Move.BCGapReset:=FALSE;
		btn_reset:=FALSE;
		s_state:=0;
END_CASE

(*触发限位开关后，相当于点击了Stop按钮*)
FTrig_ReachLS(CLK:=Unreach_LS_Far AND Unreach_LS_Near);
IF FTrig_ReachLS.Q THEN
	btn_UserGapStop:=TRUE;
END_IF
(*触发限位后，如果继续向前运动，点击move，则相当于点击stop，用于恢复move的状态位*)
IF NOT Unreach_LS_Far AND btn_UserGapMove AND UserGapPositionNew >= UserGapPositionDisplay THEN
	btn_UserGapStop:=TRUE;
END_IF
IF NOT Unreach_LS_Near AND btn_UserGapMove AND UserGapPositionNew <= UserGapPositionDisplay THEN
	btn_UserGapStop:=TRUE;
END_IF
END_ACTION

ACTION A_SpectroscopyScanningMotion:
(*输入保护*)
IF SS_Move AND SSMotionMode AND NOT RegularMotionMode THEN
	IF NOT inRange_SS_StepSize THEN
		SS_Stop:=TRUE;
		SS_Move:=FALSE;
		Error:=TRUE;
		ErrorId:=805;
		ErrorDescription:='target StepSize out of range,please check';
		RETURN;
	ELSE
		//SS_Stop:=FALSE;
		Error:=FALSE;
		ErrorId:=0;
		ErrorDescription:='';	
	END_IF
	//
	IF NOT inRange_SS_StepNumber THEN
		SS_Stop:=TRUE;
		SS_Move:=FALSE;
		Error:=TRUE;
		ErrorId:=806;
		ErrorDescription:='target StepNumber out of range,please check';
		RETURN;
	ELSE
		//SS_Stop:=FALSE;
		Error:=FALSE;
		ErrorId:=0;
		ErrorDescription:='';	
	END_IF
	IF NOT inRange_SS_StepVelocity THEN
		SS_Stop:=TRUE;
		SS_Move:=FALSE;
		Error:=TRUE;
		ErrorId:=807;
		ErrorDescription:='target StepVelocity out of range,please check';
		RETURN;
	ELSE
		//SS_Stop:=FALSE;
		Error:=FALSE;
		ErrorId:=0;
		ErrorDescription:='';	
	END_IF
	IF NOT inRange_StepEachTime_ms THEN
		SS_Stop:=TRUE;
		SS_Move:=FALSE;
		Error:=TRUE;
		ErrorId:=808;
		ErrorDescription:='target StepEachTime_ms out of range,please check';
		RETURN;
	ELSE
		//SS_Stop:=FALSE;
		Error:=FALSE;
		ErrorId:=0;
		ErrorDescription:='';	
	END_IF
END_IF
(*单步时长转换*)
StepEachTime:=INT_TO_TIME(StepEachTime_ms);
SS_TON(PT:=StepEachTime);
(*上升沿触发，初始SS位置=当前磁间隙*)
RTRG_SS_StartPositionDisplay(CLK:=SS_Move);
IF RTRG_SS_StartPositionDisplay.Q THEN
	SS_StartPositionDisplay:=UserGapPositionDisplay;
	SS_InitStartPositionDone:=TRUE;
END_IF
(*SS主程序*)
IF InitPowerDone AND InitCompensationDatasDone AND SS_Move AND SS_InitStartPositionDone THEN
	IF NOT st_Power THEN
		ErrorID:=1501;
		Error:=TRUE;
		ErrorDescription:='Plz PowerOn Frist';
		LED_Error:=TRUE;
		//btn_UserGapMove:=FALSE;
		RETURN;
	ELSE
		ErrorID:=0;
		Error:=FALSE;
		ErrorDescription:='';
		LED_Error:=FALSE;
		//btn_UserGapMove:=TRUE;
	END_IF	
CASE SS_MoveState OF
		0:
				//UserGapPositionNew:=UserGapPositionDisplay+SS_StepSize;
				UserGapPositionNew:=SS_StartPositionDisplay+SS_StepSize*(SS_currentStep+1);
				A_InitCompensationData();
				FB_Move.Mode:=5;						//1.gap;2.single;3.taper;4.debug;5.BCGap&UserMode
				FB_Move.CoupleState:=st_Couple;			
				FB_Move.PowerState:=st_Power;							
				FB_Move.BCLeftTopPosition:=LeftTopLinPositionNew;
				FB_Move.BCLeftTopVelocity:=SS_StepVelocity/2;
				FB_Move.BCRightTopPosition:=RightTopLinPositionNew;
				FB_Move.BCRightTopVelocity:=SS_StepVelocity/2;
				FB_Move.BCLeftBottomPosition:=LeftBottomLinPositionNew;
				FB_Move.BCLeftBottomVelocity:=SS_StepVelocity/2;
				FB_Move.BCRightBottomPosition:=RightBottomLinPositionNew;
				FB_Move.BCRightBottomVelocity:=SS_StepVelocity/2;		
				FB_Move.BCGapMove:=TRUE;
				FB_Move();
				SS_MoveState:=1;
		1:
				SS_TON.IN:=TRUE;
				FB_Move();
				IF FB_Move.GapMoving AND NOT SS_TimeCountBegin THEN
					SS_StepSystemTime_Begin[SS_currentStep]:=F_GetSysTime();
					SS_TimeCountBegin:=TRUE;
				END_IF
				IF NOT FB_Move.BCGapDone THEN			
					Led_Run:=TRUE;
					SS_MoveState:=1;
				ELSE									
					SS_MoveState:=66;
					SS_StepSystemTime_End[SS_currentStep]:=F_GetSysTime();
					SS_StepCountTime[SS_currentStep]:=SS_StepSystemTime_End[SS_currentStep]-SS_StepSystemTime_Begin[SS_currentStep];
					SS_TimeCountBegin:=FALSE;
				END_IF
		66:
				SS_currentStep:=SS_currentStep+1;			
				Led_Run:=FALSE;
				IF SS_currentStep=SS_StepNumber THEN								
					SS_MoveState:=88;
				END_IF
				IF SS_currentStep<SS_StepNumber THEN
					SS_MoveState:=77;
				END_IF
		77://等待单步时长够
				IF SS_TON.Q THEN
					SS_TON.IN:=FALSE;
					SS_MoveState:=0;
				END_IF
		88:
				SS_TON.IN:=FALSE;
				SS_Move:=FALSE;	
				Led_Run:=FALSE;
				SS_MoveState:=0;
				SS_currentStep:=0;
				SS_InitStartPositionDone:=FALSE;
				//SS_StepSystemTime[SS_StepNumber]:=F_GetSysTime();
	END_CASE
END_IF
(*获取每一步耗时*)
//FOR	m:= 0 TO SS_StepNumber DO
//	SS_StepCountTime[m]:=(SS_StepSystemTime_End[m]-SS_StepSystemTime_Begin[m]);
//END_FOR

(*STOP*)
IF SS_Stop OR btn_reset THEN
	FB_Move.BCGapReset:=TRUE;							(*¸øÔË¶¯FB¸øÍ£Ö¹ÐÅºÅ£¬Ê¹FB_Move×´Ì¬»Ö¸´*)
	FB_Move();											(*Æô¶¯FB_Move*)
	SS_Move:=FALSE;								(*btn_GapMove:=FALSE*)
	SS_MoveState:=0;										(*m_state:=0;*)
	CASE SS_StopState OF
			0:
				FB_Stop.Mode:=5;							(*1£ºgapÄ£Ê½£»2£ºµ¥ÁºÄ£Ê½£»3£ºtaperÄ£Ê½£»4£ºDebugÄ£Ê½£»5£ºBCGapÄ£Ê½*)
				FB_Stop.CoupleState:=st_Couple;			(*ñîºÏ×´Ì¬ÊäÈë*)
				FB_Stop.PowerState:=st_Power;				(*µçÔ´×´Ì¬ÊäÈë*)
				FB_Stop.BCGapStop:=TRUE;				(*Execute TRUE*)
				FB_Stop();								(*Æô¶¯FB*)
				SS_StopState:=1;
			1:
				FB_Stop();
				IF NOT FB_Stop.BCGapDone THEN			(*Í£Ö¹Î´Íê³É£¬Ñ­»·*)
					SS_StopState:=1;
				ELSE									(*Í£Ö¹Íê³É£¬ÏÂÒ»²½*)
					SS_StopState:=88;
				END_IF
			88:
				SS_Stop:=FALSE;						(*»Ö¸´×´Ì¬*)
				FB_Move.BCGapReset:=FALSE;				(*ÔËÐÐFB*)
				SS_StopState:=0;
				btn_reset:=FALSE;
				//SS_Stop2:=FALSE;
		END_CASE
END_IF

(*触发限位开关后，相当于点击了Stop按钮*)
FTrig_ReachLS(CLK:=Unreach_LS_Far AND Unreach_LS_Near);
IF FTrig_ReachLS.Q THEN
	SS_Stop:=TRUE;
END_IF
END_ACTION

END_PROGRAM

(* stored: Version 1.1.0.1, ProductVersion 3.1.4024.6
   POU UserMode: Id {dbb58c86-3204-4c0e-a297-03b24a68bd10}, SpecialFunc None
   Action A_CheckCoupleStatus: Id {ec531655-4226-4156-a0f2-db7d67f06866}
   Action A_CheckMotorsPos: Id {f3cd81f2-82fa-493f-8c36-20c483307c7d}
   Action A_GlobalChainProtection_EPS: Id {06b22d18-fd3c-40de-ae42-96c81b461f09}
   Action A_GlobalChainProtection_MPS: Id {214f7982-b3a1-46e2-bee6-e29b232f3cd2}
   Action A_InitCompensationData: Id {1e6a9c39-c8a5-4c48-b57c-71effe5e3747}
   Action A_MonitoringAllAxis: Id {ca11d2cd-2857-4b76-bcfc-746a563d8a76}
   Action A_OneKeyToMaxGap: Id {ba9dc3e9-1e8e-4d76-8af6-498bfc77c09c}
   Action A_PhaseLowerMotion: Id {f5505abe-8b40-4ad3-855a-7ffc19481ca9}
   Action A_PhaseLowerMotion_1: Id {69502db9-e08c-4762-acc8-458c4f879d94}
   Action A_PhaseUpperMotion: Id {b87fb803-245f-4181-b0eb-701ba9dcf58a}
   Action A_PhaseUpperMotion_1: Id {e4b83f58-f77a-4261-b358-cc7f547c3bea}
   Action A_PowerOff: Id {e3ff8ae4-6e0c-4bb4-9a62-00e47841163f}
   Action A_PowerOn: Id {cacab3c1-f169-458e-acb8-60acf8e4d140}
   Action A_RegularMotion: Id {79d2706f-89ad-4612-adf2-c80c9fc85b18}
   Action A_SpectroscopyScanningMotion: Id {6676a965-5ff1-46e4-b651-02d2762b99bc} *)
